// TIA Portal V15.1 export
// export: Created 2024-06-21T08:41:16.2567037Z, ExportSetting WithDefaults, DisplayName Totally Integrated Automation Portal, DisplayVersion V15.1 Update 5, DisplayName TIA Portal Openness, DisplayVersion V15.1 Update 5, DisplayName SINAMICS Startdrive Advanced, DisplayVersion V15.1, DisplayName G130, G150, S120, S150, SINAMICS MV, S210, DisplayVersion V15.1, DisplayName G110M, G120, G120C, G120D, G120P, DisplayVersion V15.1, DisplayName STEP 7 Professional, DisplayVersion V15.1 Update 5, DisplayName STEP 7 Safety, DisplayVersion V15.1, DisplayName WinCC Professional, DisplayVersion V15.1 Update 5, DisplayName SIMATIC Visualization Architect, DisplayVersion V15.1
FUNCTION_BLOCK "LGBRoller2W2S-MoviFitFCPN-S12B"   // FB6670, FBD
TITLE = LRoller2W2S-MoviFitFCPN / LGBRoller2W2S-MoviFitFCPN-S12B
{ S7_Optimized_Access := 'TRUE' }
AUTHOR : ENGIE
FAMILY : Transport
VERSION : 0.1
// =============================================================================
// This module is used in Applications when a roller one way two speed equipped 
// with SEW MOVIFIT-FC is needed. The roller can support single body tranport and 
// simultanious transport. The roller is equipped with a standard sensor setting, 
// one stop High Speed and one at the front for dual speed transport. The 
// roller uses standard handshaking signals to accomplish an infeed transfer 
// with the previous transport system and an outfeed with the next transport 
// system.
// The roller will support automatic Mode and manual Mode according specific 
// guidelines.
// The outfeed will be master over the infeed.
// Alarm "body not in Position" is also generated.
// All Alarms coming from sub-functions, TrfIn, TrfOut & LMotor2W2S-MoviFitFCPN or 
// from 
// local Alarm are summarized to give also the global Alarm A, B, C & D to 
// upper level.
// =============================================================================
// ============================================================================
// This module is used in Applications when a roller one way two speed equipped 
// with SEW MOVIFIT-FC is needed. The roller can support single body tranport and 
// simultanious transport. The roller is equipped with a standard sensor setting, 
// one stop High Speed and one at the front for dual speed transport. The 
// roller uses standard handshaking signals to accomplish an infeed transfer 
// with the previous transport system and an outfeed with the next transport 
// system.
// The roller will support automatic Mode and manual Mode according specific 
// guidelines.
// The outfeed will be master over the infeed.
// Alarm "body not in Position" is also generated.
// All Alarms coming from sub-functions, TrfIn, TrfOut & LMotor2W2S-MoviFitFCPN or 
// from 
// local Alarm are summarized to give also the global Alarm A, B, C & D to 
// upper level.
// ============================================================================
// stored: AutoNumber false, IsIECCheckEnabled false, IsRetainMemResEnabled false, MemoryReserve 100, SetENOAutomatically False, UDAEnableTagReadback false
   VAR_INPUT
      I_StopDetSet { ExternalAccessible := 'False'; ExternalVisible := 'False'; ExternalWritable := 'False'} : Bool;   // Stop detection set
      I_LowSpeedDetSet { ExternalAccessible := 'False'; ExternalVisible := 'False'; ExternalWritable := 'False'} : Bool;   // Lowspeed detection set
      I_StopDetRes { ExternalAccessible := 'False'; ExternalVisible := 'False'; ExternalWritable := 'False'} : Bool;   // Stop detection Reset
      I_LowSpeedDetRes { ExternalAccessible := 'False'; ExternalVisible := 'False'; ExternalWritable := 'False'} : Bool;   // Lowspeed stop detection Reset
      I_OccupiedDet { ExternalAccessible := 'False'; ExternalVisible := 'False'; ExternalWritable := 'False'} : Bool;   // Occupied detection
      I_TrfInSetBegin { ExternalAccessible := 'False'; ExternalVisible := 'False'; ExternalWritable := 'False'} : Bool;   // Load Begin: condition to start transfer IN set
      I_TrfInSetIntlkOk { ExternalAccessible := 'False'; ExternalVisible := 'False'; ExternalWritable := 'False'} : Bool;   // Transfer IN Interlock Set OK
      I_TrfInResBegin { ExternalAccessible := 'False'; ExternalVisible := 'False'; ExternalWritable := 'False'} : Bool;   // Load Begin: condition to start transfer IN Reset
      I_TrfInResIntlkOk { ExternalAccessible := 'False'; ExternalVisible := 'False'; ExternalWritable := 'False'} : Bool;   // Transfer IN Interlock Reset OKt
      I_TrfOutSetBegin { ExternalAccessible := 'False'; ExternalVisible := 'False'; ExternalWritable := 'False'} : Bool;   // Unload Begin: condition to start transfer OUT set
      I_TrfOutSetIntlkOk { ExternalAccessible := 'False'; ExternalVisible := 'False'; ExternalWritable := 'False'} : Bool;   // Transfer Out Interlock Set Ok
      I_TrfOutResBegin { ExternalAccessible := 'False'; ExternalVisible := 'False'; ExternalWritable := 'False'} : Bool;   // Unload Begin: condition to start transfer OUT Reset
      I_TrfOutResIntlkOk { ExternalAccessible := 'False'; ExternalVisible := 'False'; ExternalWritable := 'False'} : Bool;   // Transfer OUT Interlock Reset Ok
      I_TrfInSetRdyDlv { ExternalAccessible := 'False'; ExternalVisible := 'False'; ExternalWritable := 'False'} : Bool;   // Ready to deliver: Signal from previous object set
      I_TrfInSetTM { ExternalAccessible := 'False'; ExternalVisible := 'False'; ExternalWritable := 'False'} : Bool;   // Transfer busy signal from previous equipement set
      I_TrfOutSetRdyRcv { ExternalAccessible := 'False'; ExternalVisible := 'False'; ExternalWritable := 'False'} : Bool;   // Ready to Receive: Signal from next object set
      I_TrfOutSetArrived { ExternalAccessible := 'False'; ExternalVisible := 'False'; ExternalWritable := 'False'} : Bool;   // Body Arrived: Signal from next object Set
      I_TrfInResRdyDlv { ExternalAccessible := 'False'; ExternalVisible := 'False'; ExternalWritable := 'False'} : Bool;   // Ready to deliver: Signal from previous object Reset
      I_TrfInResTM { ExternalAccessible := 'False'; ExternalVisible := 'False'; ExternalWritable := 'False'} : Bool;   // Transfer busy signal from previous equipement Reset
      I_TrfOutResRdyRcv { ExternalAccessible := 'False'; ExternalVisible := 'False'; ExternalWritable := 'False'} : Bool;   // Ready to Receive: Signal from next object Reset
      I_TrfOutResArrived { ExternalAccessible := 'False'; ExternalVisible := 'False'; ExternalWritable := 'False'} : Bool;   // Body Arrived: Signal from next object Reset
      I_ManInfeedAllowedSet { ExternalAccessible := 'False'; ExternalVisible := 'False'; ExternalWritable := 'False'} : Bool;   // Manual Infeed Allowed Set (without PushButton)
      I_ManInfeedAllowedRes { ExternalAccessible := 'False'; ExternalVisible := 'False'; ExternalWritable := 'False'} : Bool;   // Manual Infeed Allowed Reset (without PushButton)
      I_ManLowSpdSel { ExternalAccessible := 'False'; ExternalVisible := 'False'; ExternalWritable := 'False'} : Bool;   // Low speed Selected in manual / Low speed Selected in manual by other roller
      I_ManHighSpdSel { ExternalAccessible := 'False'; ExternalVisible := 'False'; ExternalWritable := 'False'} : Bool;   // Low speed Selected in manual / High speed Selected in manual by other roller
      I_MotorProtection { ExternalAccessible := 'False'; ExternalVisible := 'False'; ExternalWritable := 'False'} : Bool;   // Motorprotection
      I_ReleaseBrake { ExternalAccessible := 'False'; ExternalVisible := 'False'; ExternalWritable := 'False'} : Bool;   // Release brake
      I_LocalPBSet { ExternalAccessible := 'False'; ExternalVisible := 'False'; ExternalWritable := 'False'} : Bool;   // Push button for manual movememt (on local panel)
      I_LocalPBRes { ExternalAccessible := 'False'; ExternalVisible := 'False'; ExternalWritable := 'False'} : Bool;   // Push button for manual movememt Reset(on local panel)
      I_BeltControlSetDet { ExternalAccessible := 'False'; ExternalVisible := 'False'; ExternalWritable := 'False'} : Bool;   // Sensor Belt Control Roller Set Direction
      I_BeltControlResDet { ExternalAccessible := 'False'; ExternalVisible := 'False'; ExternalWritable := 'False'} : Bool;   // Sensor Belt Control Roller Res Direction
      I_SafetyOk { ExternalAccessible := 'False'; ExternalVisible := 'False'; ExternalWritable := 'False'} : Bool;   // Safety Ok
      I_MotionStopOk { ExternalAccessible := 'False'; ExternalVisible := 'False'; ExternalWritable := 'False'} : Bool;   // Safety Ok / The motion stop is Ok
      I_LowSpeed { ExternalAccessible := 'False'; ExternalVisible := 'False'; ExternalWritable := 'False'} : Real;   // Low speed Value (set-up %)
      I_HighSpeed { ExternalAccessible := 'False'; ExternalVisible := 'False'; ExternalWritable := 'False'} : Real;   // High speed Value (set-up %)
      I_SafetyStatusWord1 { ExternalAccessible := 'False'; ExternalVisible := 'False'; ExternalWritable := 'False'} : Word;   // Safety Status / Safety Status Word
      I_SafetyStatusWord2 { ExternalAccessible := 'False'; ExternalVisible := 'False'; ExternalWritable := 'False'} : Word;   // Safety Status / Safety Status Word
      I_SafetyStatusWord3 { ExternalAccessible := 'False'; ExternalVisible := 'False'; ExternalWritable := 'False'} : Word;   // Safety Status / Safety Status Word
      I_SafetyControlWord1 { ExternalAccessible := 'False'; ExternalVisible := 'False'; ExternalWritable := 'False'} : Word;   // Safety Control Word
      I_SafetyControlWord2 { ExternalAccessible := 'False'; ExternalVisible := 'False'; ExternalWritable := 'False'} : Word;   // Safety Control Word
   END_VAR
   VAR_OUTPUT
      O_ReleaseBrake { ExternalAccessible := 'False'; ExternalVisible := 'False'; ExternalWritable := 'False'} : Bool;   // Release the brake of the Motor
      O_Active { ExternalAccessible := 'False'; ExternalVisible := 'False'; ExternalWritable := 'False'} : Bool;   // Roller is Active
      O_TrfInSetRdyRcv { ExternalAccessible := 'False'; ExternalVisible := 'False'; ExternalWritable := 'False'} : Bool;   // Ready to Receive: Signal to previous object set
      O_TrfInSetArrived { ExternalAccessible := 'False'; ExternalVisible := 'False'; ExternalWritable := 'False'} : Bool;   // Body Arrived: Signal to previous object Set
      O_TrfOutSetRdyDlv { ExternalAccessible := 'False'; ExternalVisible := 'False'; ExternalWritable := 'False'} : Bool;   // Ready to Deliver: Signal to next object set
      O_TrfOutSetTM { ExternalAccessible := 'False'; ExternalVisible := 'False'; ExternalWritable := 'False'} : Bool;   // Transfer: Signal to next object set
      O_TrfInResRdyRcv { ExternalAccessible := 'False'; ExternalVisible := 'False'; ExternalWritable := 'False'} : Bool;   // Ready to Receive: Signal to previous object Reset
      O_TrfInResArrived { ExternalAccessible := 'False'; ExternalVisible := 'False'; ExternalWritable := 'False'} : Bool;   // Body Arrived: Signal to previous object Reset
      O_TrfOutResRdyDlv { ExternalAccessible := 'False'; ExternalVisible := 'False'; ExternalWritable := 'False'} : Bool;   // Ready to Deliver: Signal to next object Reset
      O_TrfOutResTM { ExternalAccessible := 'False'; ExternalVisible := 'False'; ExternalWritable := 'False'} : Bool;   // Transfer: Signal to next object Reset
      O_TrfInSetActive { ExternalAccessible := 'False'; ExternalVisible := 'False'; ExternalWritable := 'False'} : Bool;   // Transfer in set active
      O_TrfInSetFinished { ExternalAccessible := 'False'; ExternalVisible := 'False'; ExternalWritable := 'False'} : Bool;   // Transfer in set finished
      O_TrfOutSetActive { ExternalAccessible := 'False'; ExternalVisible := 'False'; ExternalWritable := 'False'} : Bool;   // Transfer out set active
      O_TrfOutSetFinished { ExternalAccessible := 'False'; ExternalVisible := 'False'; ExternalWritable := 'False'} : Bool;   // Transfer out set finished
      O_TrfInResActive { ExternalAccessible := 'False'; ExternalVisible := 'False'; ExternalWritable := 'False'} : Bool;   // Transfer in Reset active
      O_TrfInResFinished { ExternalAccessible := 'False'; ExternalVisible := 'False'; ExternalWritable := 'False'} : Bool;   // Transfer in Reset finished
      O_TrfOutResActive { ExternalAccessible := 'False'; ExternalVisible := 'False'; ExternalWritable := 'False'} : Bool;   // Transfer out Reset active
      O_TrfOutResFinished { ExternalAccessible := 'False'; ExternalVisible := 'False'; ExternalWritable := 'False'} : Bool;   // Transfer out Reset finished
      O_BodyInPosition { ExternalAccessible := 'False'; ExternalVisible := 'False'; ExternalWritable := 'False'} : Bool;   // Body in Position on roller
      O_ManLowSpdSel { ExternalAccessible := 'False'; ExternalVisible := 'False'; ExternalWritable := 'False'} : Bool;   // Low speed Selected in manual
      O_ManHighSpdSel { ExternalAccessible := 'False'; ExternalVisible := 'False'; ExternalWritable := 'False'} : Bool;   // Low speed Selected in manual / High speed Selected in manual
      O_LedRoller { ExternalAccessible := 'False'; ExternalVisible := 'False'; ExternalWritable := 'False'} : Bool;   // Led of roller
      O_LSpdSetMotorCmd { ExternalAccessible := 'False'; ExternalVisible := 'False'; ExternalWritable := 'False'} : Bool;   // Low Speed Set Command from function after Interlock
      O_HSpdSetMotorCmd { ExternalAccessible := 'False'; ExternalVisible := 'False'; ExternalWritable := 'False'} : Bool;   // High Speed Set Command from function after Interlock
      O_LSpdResMotorCmd { ExternalAccessible := 'False'; ExternalVisible := 'False'; ExternalWritable := 'False'} : Bool;   // Low speed Reset Command from function after Interlock
      O_HSpdResMotorCmd { ExternalAccessible := 'False'; ExternalVisible := 'False'; ExternalWritable := 'False'} : Bool;   // High speed Reset Command from function after Interlock
      O_AlarmABCondition { ExternalAccessible := 'False'; ExternalVisible := 'False'; ExternalWritable := 'False'} : Bool;   // Alarm AB Condition
      O_AlarmA { ExternalAccessible := 'False'; ExternalVisible := 'False'; ExternalWritable := 'False'} : Bool;   // Alarm A
      O_AlarmB { ExternalAccessible := 'False'; ExternalVisible := 'False'; ExternalWritable := 'False'} : Bool;   // Alarm B
      O_AlarmC { ExternalAccessible := 'False'; ExternalVisible := 'False'; ExternalWritable := 'False'} : Bool;   // Alarm C
      O_AlarmD { ExternalAccessible := 'False'; ExternalVisible := 'False'; ExternalWritable := 'False'} : Bool;   // Alarm D
      O_Occupied { ExternalAccessible := 'False'; ExternalVisible := 'False'; ExternalWritable := 'False'} : Bool;   // Roller Occupied
      H_AlarmDWord { ExternalAccessible := 'False'; ExternalVisible := 'False'; ExternalWritable := 'False'} : DWord;   // Alarm Word
   END_VAR
   VAR_IN_OUT
      IO_Modes : "Modes";   // Modes
      H_HMI : "H_HMI";   // Animation
      "H_GBRoller2W2S-MoviFitFCPN-S12B" : "H_GBRoller2W2S-MoviFitFCPN-S12B";   // Animation
      C_RollerConvConfig : "RollerConvMoviFitFCPNConfig";   // Config
   END_VAR
   VAR
      _LTrfInSet { ExternalAccessible := 'False'; ExternalVisible := 'False'; ExternalWritable := 'False'} : "LGBTrfIn";   // FB
      _LTrfOutSet { ExternalAccessible := 'False'; ExternalVisible := 'False'; ExternalWritable := 'False'} : "LGBTrfOut";   // FB
      _LTrfInRes { ExternalAccessible := 'False'; ExternalVisible := 'False'; ExternalWritable := 'False'} : "LGBTrfIn";   // FB
      _LTrfOutRes { ExternalAccessible := 'False'; ExternalVisible := 'False'; ExternalWritable := 'False'} : "LGBTrfOut";   // FB
      _Motor { ExternalAccessible := 'False'; ExternalVisible := 'False'; ExternalWritable := 'False'} : "LGBMotor2W2S-MoviFitFCPN-S12B";   // FB
      AB_BeltControlSetDet { ExternalAccessible := 'False'; ExternalVisible := 'False'; ExternalWritable := 'False'} : Bool;   // Belt Check Roller Set Direction
      AB_BeltControlResDet { ExternalAccessible := 'False'; ExternalVisible := 'False'; ExternalWritable := 'False'} : Bool;   // Belt Check Roller Reset Direction
      AC_BodyNotInPos { ExternalAccessible := 'False'; ExternalVisible := 'False'; ExternalWritable := 'False'} : Bool;   // Body, Skid Not In Position
      AD_TrfInResInterlock { ExternalAccessible := 'False'; ExternalVisible := 'False'; ExternalWritable := 'False'} : Bool;   // Interlock Not Ok Transport In Reset
      AB_TrfOutSetOverTime { ExternalAccessible := 'False'; ExternalVisible := 'False'; ExternalWritable := 'False'} : Bool;   // Timeout Set
      AD_TrfOutSetInterlock { ExternalAccessible := 'False'; ExternalVisible := 'False'; ExternalWritable := 'False'} : Bool;   // Interlock Not Ok Transport Out Set
      AD_TrfInSetInterlock { ExternalAccessible := 'False'; ExternalVisible := 'False'; ExternalWritable := 'False'} : Bool;   // Interlock Not Ok Transport In Set
      AB_TrfOutResOverTime { ExternalAccessible := 'False'; ExternalVisible := 'False'; ExternalWritable := 'False'} : Bool;   // Timeout Reset
      AD_TrfOutResInterlock { ExternalAccessible := 'False'; ExternalVisible := 'False'; ExternalWritable := 'False'} : Bool;   // Interlock Not Ok Transport Out Reset
      AB_LSpeedDetMissing { ExternalAccessible := 'False'; ExternalVisible := 'False'; ExternalWritable := 'False'} : Bool;   // Low Speed Detector Missing
      AA_MotorProtection { ExternalAccessible := 'False'; ExternalVisible := 'False'; ExternalWritable := 'False'} : Bool;   // Motorprotection Tripped / Motor Protection Tripped
      AA_SafetySwitch { ExternalAccessible := 'False'; ExternalVisible := 'False'; ExternalWritable := 'False'} : Bool;   // Safety Switch Not Ok
      AB_STO { ExternalAccessible := 'False'; ExternalVisible := 'False'; ExternalWritable := 'False'} : Bool;   // Safety Switch Not Ok / Safety output to drive is active but no response from drive that the safety is ok
      AD_Warning { ExternalAccessible := 'False'; ExternalVisible := 'False'; ExternalWritable := 'False'} : Bool;   // Frequency Control
      AA_NoBusControl { ExternalAccessible := 'False'; ExternalVisible := 'False'; ExternalWritable := 'False'} : Bool;   // Frequency Control / Bus control inactive / Frekvensstyrning
      AB_Alarm { ExternalAccessible := 'False'; ExternalVisible := 'False'; ExternalWritable := 'False'} : Bool;   // Frequency Control
      AC_TrfInStopped { ExternalAccessible := 'False'; ExternalVisible := 'False'; ExternalWritable := 'False'} : Bool;   // Transfer In Stopped
      AC_StopDetSet { ExternalAccessible := 'False'; ExternalVisible := 'False'; ExternalWritable := 'False'} : Bool;   // Body, Skid Not In Position Stop Det Set
      AC_StopDetRes { ExternalAccessible := 'False'; ExternalVisible := 'False'; ExternalWritable := 'False'} : Bool;   // Body, Skid Not In Position Stop Det Reset
      AC_LowSpdDetSet { ExternalAccessible := 'False'; ExternalVisible := 'False'; ExternalWritable := 'False'} : Bool;   // Body, Skid Not In Position Low Speed Det Set
      AC_LowSpdDetRes { ExternalAccessible := 'False'; ExternalVisible := 'False'; ExternalWritable := 'False'} : Bool;   // Body, Skid Not In Position Low Speed Det Reset
      AD_MotionStop { ExternalAccessible := 'False'; ExternalVisible := 'False'; ExternalWritable := 'False'} : Bool;   // Motion Stop
      AC_ConfigCalibrationAlm { ExternalAccessible := 'False'; ExternalVisible := 'False'; ExternalWritable := 'False'} : Bool;   // The Config values for Alarm Transfer time must be ALL zero or ALL different from zero
      AD_CalibrationSetWarn { ExternalAccessible := 'False'; ExternalVisible := 'False'; ExternalWritable := 'False'} : Bool;   // No High speed selected so Calibration is not possible for SET direction
      AD_CalibrationResetWarn { ExternalAccessible := 'False'; ExternalVisible := 'False'; ExternalWritable := 'False'} : Bool;   // No High speed selected so Calibration is not possible for RESET direction
      AC_ConfigRampAlm { ExternalAccessible := 'False'; ExternalVisible := 'False'; ExternalWritable := 'False'} : Bool;   // The config value for the ramp is not correct, must be zero or the config values for the calculation of the ramp must be ALL zero
      AC_ConfigRampCalcAlm { ExternalAccessible := 'False'; ExternalVisible := 'False'; ExternalWritable := 'False'} : Bool;   // The config values for the calculation of the ramp must be ALL different from zero
      PODataNotEnabled { ExternalAccessible := 'False'; ExternalVisible := 'False'; ExternalWritable := 'False'} : Bool;   // Bus control inactive
      SafetyOk { ExternalAccessible := 'False'; ExternalVisible := 'False'; ExternalWritable := 'False'} : Bool;   // Safety Ok
   END_VAR
   VAR RETAIN
      LowSpeedSetDetOk { ExternalAccessible := 'False'; ExternalVisible := 'False'; ExternalWritable := 'False'} : Bool;   // Low speed detector set ok
      LowSpeedResDetOk { ExternalAccessible := 'False'; ExternalVisible := 'False'; ExternalWritable := 'False'} : Bool;   // Low speed detector Reset ok
   END_VAR
   VAR
      AllDet { ExternalAccessible := 'False'; ExternalVisible := 'False'; ExternalWritable := 'False'} : Bool;   // AND of all detections
      AnyDet { ExternalAccessible := 'False'; ExternalVisible := 'False'; ExternalWritable := 'False'} : Bool;   // OR of all detections
      MotorLoopActive { ExternalAccessible := 'False'; ExternalVisible := 'False'; ExternalWritable := 'False'} : Bool;   // Motor Loop Active
      TrfInSetIntlkOk { ExternalAccessible := 'False'; ExternalVisible := 'False'; ExternalWritable := 'False'} : Bool;   // Transfer IN Interlock Set OK
      TrfInResIntlkOk { ExternalAccessible := 'False'; ExternalVisible := 'False'; ExternalWritable := 'False'} : Bool;   // Transfer IN Interlock Reset OKt / Transfer IN Interlock Reset OK
      TrfOutResIntlkOk { ExternalAccessible := 'False'; ExternalVisible := 'False'; ExternalWritable := 'False'} : Bool;   // Transfer OUT Interlock Reset Ok
      TrfOutSetIntlkOk { ExternalAccessible := 'False'; ExternalVisible := 'False'; ExternalWritable := 'False'} : Bool;   // Transfer Out Interlock Set Ok
      TrfInResCmd { ExternalAccessible := 'False'; ExternalVisible := 'False'; ExternalWritable := 'False'} : Bool;   // Command after Interlock to Motor Reset
      TrfInfeedHoldSet { ExternalAccessible := 'False'; ExternalVisible := 'False'; ExternalWritable := 'False'} : Bool;   // Transfer infeed hold set direction
      TrfOutSetCmd { ExternalAccessible := 'False'; ExternalVisible := 'False'; ExternalWritable := 'False'} : Bool;   // Command after Interlock to Motor set
      TrfOutfeedHoldSet { ExternalAccessible := 'False'; ExternalVisible := 'False'; ExternalWritable := 'False'} : Bool;   // Transfer outfeed hold set direction
      TrfInSetCmd { ExternalAccessible := 'False'; ExternalVisible := 'False'; ExternalWritable := 'False'} : Bool;   // Command after Interlock to Motor set
      TrfInfeedHoldRes { ExternalAccessible := 'False'; ExternalVisible := 'False'; ExternalWritable := 'False'} : Bool;   // Transfer infeed hold Reset direction
      TrfOutResCmd { ExternalAccessible := 'False'; ExternalVisible := 'False'; ExternalWritable := 'False'} : Bool;   // Command after Interlock to Motor Reset
      TrfOutfeedHoldRes { ExternalAccessible := 'False'; ExternalVisible := 'False'; ExternalWritable := 'False'} : Bool;   // Transfer outfeed hold Reset direction
      MotorCmdLSpdSet { ExternalAccessible := 'False'; ExternalVisible := 'False'; ExternalWritable := 'False'} : Bool;   // Command to Motorloop low Speed Set
      MotorCmdLSpdRes { ExternalAccessible := 'False'; ExternalVisible := 'False'; ExternalWritable := 'False'} : Bool;   // Command to Motorloop low speed Reset
      MotorCmdHSpdSet { ExternalAccessible := 'False'; ExternalVisible := 'False'; ExternalWritable := 'False'} : Bool;   // Command to Motorloop High Speed Set
      MotorCmdHSpdRes { ExternalAccessible := 'False'; ExternalVisible := 'False'; ExternalWritable := 'False'} : Bool;   // Command to Motorloop High Speed Reset
   END_VAR
   VAR RETAIN
      LowSpeedDetSetMem { ExternalAccessible := 'False'; ExternalVisible := 'False'; ExternalWritable := 'False'} : Bool;   // Memorisation stop High Speed Set direction
      LowSpeedDetResMem { ExternalAccessible := 'False'; ExternalVisible := 'False'; ExternalWritable := 'False'} : Bool;   // Memorisation stop high peed Reset direction
   END_VAR
   VAR
      TrfInSetActive { ExternalAccessible := 'False'; ExternalVisible := 'False'; ExternalWritable := 'False'} : Bool;   // Load Active Set
      TrfOutSetActive { ExternalAccessible := 'False'; ExternalVisible := 'False'; ExternalWritable := 'False'} : Bool;   // Unload active Set
      TrfOutSetFinished { ExternalAccessible := 'False'; ExternalVisible := 'False'; ExternalWritable := 'False'} : Bool;   // Unload finished Set
      TrfInResActive { ExternalAccessible := 'False'; ExternalVisible := 'False'; ExternalWritable := 'False'} : Bool;   // Load Active Reset
      TrfOutResActive { ExternalAccessible := 'False'; ExternalVisible := 'False'; ExternalWritable := 'False'} : Bool;   // Unload active Reset
      TrfOutResFinished { ExternalAccessible := 'False'; ExternalVisible := 'False'; ExternalWritable := 'False'} : Bool;   // Unload finished Reset
      StationOnly { ExternalAccessible := 'False'; ExternalVisible := 'False'; ExternalWritable := 'False'} : Bool;   // Station Only
      AlarmA { ExternalAccessible := 'False'; ExternalVisible := 'False'; ExternalWritable := 'False'} : Bool;   // Alarm A
      AlarmB { ExternalAccessible := 'False'; ExternalVisible := 'False'; ExternalWritable := 'False'} : Bool;   // Alarm B
      AlarmC { ExternalAccessible := 'False'; ExternalVisible := 'False'; ExternalWritable := 'False'} : Bool;   // Alarm C
      AlarmD { ExternalAccessible := 'False'; ExternalVisible := 'False'; ExternalWritable := 'False'} : Bool;   // Alarm D
      AlarmABCondition { ExternalAccessible := 'False'; ExternalVisible := 'False'; ExternalWritable := 'False'} : Bool;   // Alarm AB Condition
      ManLowSpdSel { ExternalAccessible := 'False'; ExternalVisible := 'False'; ExternalWritable := 'False'} : Bool;   // Low speed Selected in manual
      BodyInPosition { ExternalAccessible := 'False'; ExternalVisible := 'False'; ExternalWritable := 'False'} : Bool;   // Body in Position
      TrfInResRdyRcv { ExternalAccessible := 'False'; ExternalVisible := 'False'; ExternalWritable := 'False'} : Bool;   // Ready to Receive: Signal to previous object Reset
      TrfInResArrived { ExternalAccessible := 'False'; ExternalVisible := 'False'; ExternalWritable := 'False'} : Bool;   // Body Arrived: Signal to previous object Reset
      TrfInResFinished { ExternalAccessible := 'False'; ExternalVisible := 'False'; ExternalWritable := 'False'} : Bool;   // Body Arrived: Signal to TrfOut module Reset (Reset TrfOutCmd)
      TrfOutSetRdyDlv { ExternalAccessible := 'False'; ExternalVisible := 'False'; ExternalWritable := 'False'} : Bool;   // Ready to Deliver: Signal to next object set
      TrfOutSetTM { ExternalAccessible := 'False'; ExternalVisible := 'False'; ExternalWritable := 'False'} : Bool;   // Transfer : Signal transfer memory to next object set
      TrfInSetTrfOutSetTM { ExternalAccessible := 'False'; ExternalVisible := 'False'; ExternalWritable := 'False'} : Bool;   // Transfer memory set
      TrfInSetRdyRcv { ExternalAccessible := 'False'; ExternalVisible := 'False'; ExternalWritable := 'False'} : Bool;   // Ready to Receive: Signal to previous object set
      TrfInSetArrived { ExternalAccessible := 'False'; ExternalVisible := 'False'; ExternalWritable := 'False'} : Bool;   // Body Arrived: Signal to previous object Set
      TrfInSetFinished { ExternalAccessible := 'False'; ExternalVisible := 'False'; ExternalWritable := 'False'} : Bool;   // Body Arrived: Signal to TrfOut module set (Reset TrfOutCmd)
      StopTrfOutSetCmd { ExternalAccessible := 'False'; ExternalVisible := 'False'; ExternalWritable := 'False'} : Bool;   // Body Arrived: Signal to previous object Set
      TrfOutResRdyDlv { ExternalAccessible := 'False'; ExternalVisible := 'False'; ExternalWritable := 'False'} : Bool;   // Ready to Deliver: Signal to next object Reset
      TrfOutResTM { ExternalAccessible := 'False'; ExternalVisible := 'False'; ExternalWritable := 'False'} : Bool;   // Transfer : Signal transfer memory to next object Reset
      TrfInResTrfOutResTM { ExternalAccessible := 'False'; ExternalVisible := 'False'; ExternalWritable := 'False'} : Bool;   // Transfer memory Reset
      MotorLoopAlarmCond { ExternalAccessible := 'False'; ExternalVisible := 'False'; ExternalWritable := 'False'} : Bool;   // Motor loop Alarm condition
      TrfOutResAlmCond { ExternalAccessible := 'False'; ExternalVisible := 'False'; ExternalWritable := 'False'} : Bool;   // TrfOut Alarm condition
      TrfOutSetAlmCond { ExternalAccessible := 'False'; ExternalVisible := 'False'; ExternalWritable := 'False'} : Bool;   // TrfOut Alarm condition
      StopTrfOutResCmd { ExternalAccessible := 'False'; ExternalVisible := 'False'; ExternalWritable := 'False'} : Bool;   // Body Arrived: Signal to previous object Reset
      LowSpeedDetMisingCond { ExternalAccessible := 'False'; ExternalVisible := 'False'; ExternalWritable := 'False'} : Bool;   // Low speed detector misiing condition
      ReleaseBrake { ExternalAccessible := 'False'; ExternalVisible := 'False'; ExternalWritable := 'False'} : Bool;   // Release brake
      ReadyForOperation { ExternalAccessible := 'False'; ExternalVisible := 'False'; ExternalWritable := 'False'} : Bool;   // Ready for operation
      BeltControlSetAlarmABCondition { ExternalAccessible := 'False'; ExternalVisible := 'False'; ExternalWritable := 'False'} : Bool;   // Belt Control AB Condition
      BeltControlResAlarmABCondition { ExternalAccessible := 'False'; ExternalVisible := 'False'; ExternalWritable := 'False'} : Bool;   // Belt Control AB Condition
      _BeltControlSet { ExternalAccessible := 'False'; ExternalVisible := 'False'; ExternalWritable := 'False'} : "L1AlarmMultiIn";   // FB
      _BeltControlRes { ExternalAccessible := 'False'; ExternalVisible := 'False'; ExternalWritable := 'False'} : "L1AlarmMultiIn";   // FB
      BeltPulseCountSet { ExternalAccessible := 'False'; ExternalVisible := 'False'; ExternalWritable := 'False'} : DInt;   // Temp
      BeltPulseCountRes { ExternalAccessible := 'False'; ExternalVisible := 'False'; ExternalWritable := 'False'} : DInt;   // Temp
      _InitBeltCntSet { ExternalAccessible := 'False'; ExternalVisible := 'False'; ExternalWritable := 'False'} : "LChangeOfState";   // FB
      _InitBeltCntRes { ExternalAccessible := 'False'; ExternalVisible := 'False'; ExternalWritable := 'False'} : "LChangeOfState";   // FB
      BeltPosEdgeSet1 { ExternalAccessible := 'False'; ExternalVisible := 'False'; ExternalWritable := 'False'} : Bool;   // Pos Edge
      BeltPosEdgeSet2 { ExternalAccessible := 'False'; ExternalVisible := 'False'; ExternalWritable := 'False'} : Bool;   // Pos Edge
      BeltPosEdgeRes1 { ExternalAccessible := 'False'; ExternalVisible := 'False'; ExternalWritable := 'False'} : Bool;   // Pos Edge
      BeltPosEdgeRes2 { ExternalAccessible := 'False'; ExternalVisible := 'False'; ExternalWritable := 'False'} : Bool;   // Pos Edge
      InitBeltCounterSet { ExternalAccessible := 'False'; ExternalVisible := 'False'; ExternalWritable := 'False'} : Bool;   // Init
      InitBeltCounterRes { ExternalAccessible := 'False'; ExternalVisible := 'False'; ExternalWritable := 'False'} : Bool;   // Init
      _StationOnly { ExternalAccessible := 'False'; ExternalVisible := 'False'; ExternalWritable := 'False'} : "LToggle";   // FB
      _NoTrfIn { ExternalAccessible := 'False'; ExternalVisible := 'False'; ExternalWritable := 'False'} : "LToggle";   // FB
      Edge { ExternalAccessible := 'False'; ExternalVisible := 'False'; ExternalWritable := 'False'} : Array[1..7] of Bool;   // Edge
   END_VAR
   VAR_TEMP
      NotUsedH_HMI : "H_HMI";   // Temp
      H_HMITrfInSet : "H_HMI";   // Temp
      H_HMITrfInRes : "H_HMI";   // Temp
      H_HMITrfOutSet : "H_HMI";   // Temp
      H_HMITrfOutRes : "H_HMI";   // Temp
      H_HMIMotor : "H_HMI";   // Temp
      HMICMD : "ConvHMICMD";   // Temp
      TempDInt : DInt;   // Temp DInt
   END_VAR
   VAR_TEMP   // added for the SCL form of the ladder/FBD networks
      _w1 : Bool;
      _w2 : Bool;
      _w3 : Bool;
      _w4 : Bool;
   END_VAR
BEGIN

REGION Network 1: **** 1 - Inputs **** HMI Commands
   // HMI Commands
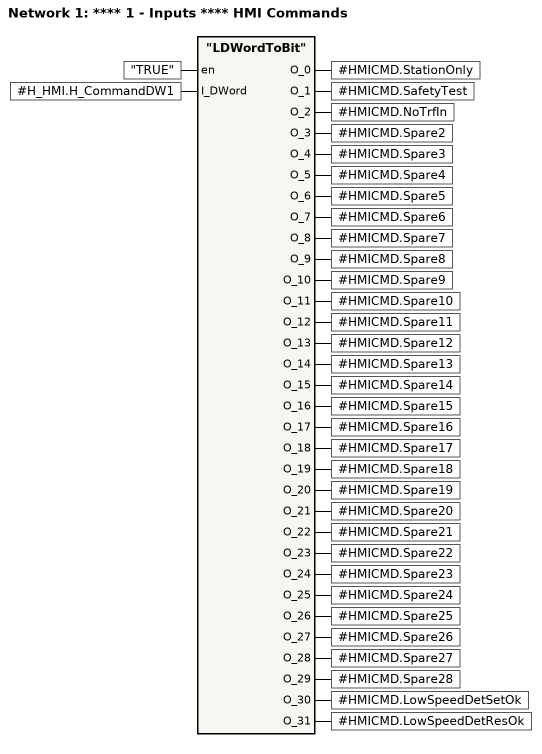
   IF "TRUE" THEN
       "LDWordToBit"(I_DWord := #H_HMI.H_CommandDW1,
                     O_0 => #HMICMD.StationOnly,
                     O_1 => #HMICMD.SafetyTest,
                     O_2 => #HMICMD.NoTrfIn,
                     O_3 => #HMICMD.Spare2,
                     O_4 => #HMICMD.Spare3,
                     O_5 => #HMICMD.Spare4,
                     O_6 => #HMICMD.Spare5,
                     O_7 => #HMICMD.Spare6,
                     O_8 => #HMICMD.Spare7,
                     O_9 => #HMICMD.Spare8,
                     O_10 => #HMICMD.Spare9,
                     O_11 => #HMICMD.Spare10,
                     O_12 => #HMICMD.Spare11,
                     O_13 => #HMICMD.Spare12,
                     O_14 => #HMICMD.Spare13,
                     O_15 => #HMICMD.Spare14,
                     O_16 => #HMICMD.Spare15,
                     O_17 => #HMICMD.Spare16,
                     O_18 => #HMICMD.Spare17,
                     O_19 => #HMICMD.Spare18,
                     O_20 => #HMICMD.Spare19,
                     O_21 => #HMICMD.Spare20,
                     O_22 => #HMICMD.Spare21,
                     O_23 => #HMICMD.Spare22,
                     O_24 => #HMICMD.Spare23,
                     O_25 => #HMICMD.Spare24,
                     O_26 => #HMICMD.Spare25,
                     O_27 => #HMICMD.Spare26,
                     O_28 => #HMICMD.Spare27,
                     O_29 => #HMICMD.Spare28,
                     O_30 => #HMICMD.LowSpeedDetSetOk,
                     O_31 => #HMICMD.LowSpeedDetResOk);
   END_IF;
END_REGION

REGION Network 2: **** 1 - Inputs **** AND of all detections
   // AND of all detections
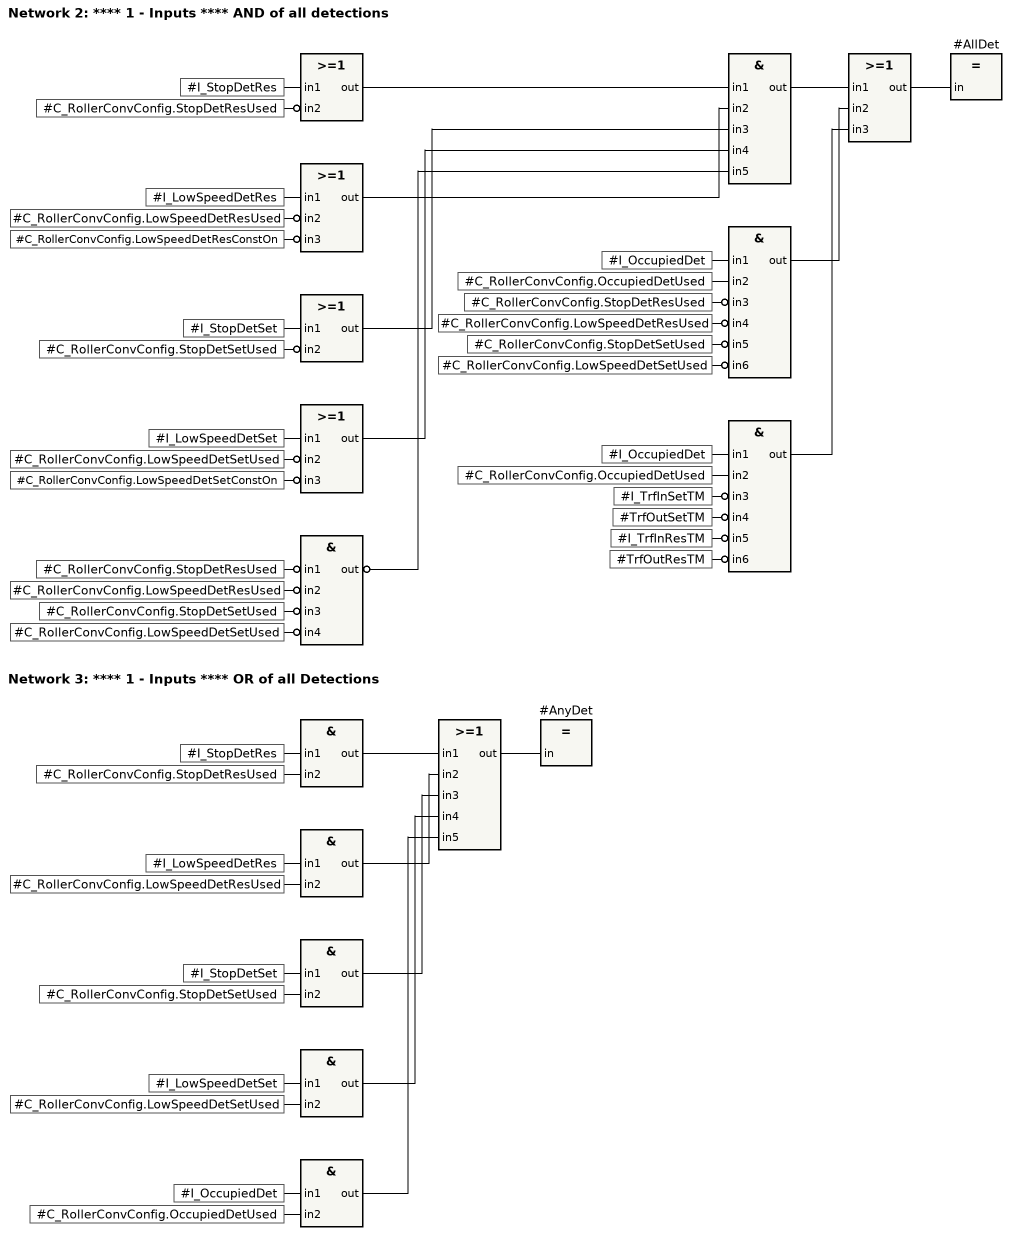
   #AllDet := ((#I_StopDetRes OR NOT #C_RollerConvConfig.StopDetResUsed) AND (#I_LowSpeedDetRes OR NOT #C_RollerConvConfig.LowSpeedDetResUsed OR NOT #C_RollerConvConfig.LowSpeedDetResConstOn) AND (#I_StopDetSet OR NOT #C_RollerConvConfig.StopDetSetUsed) AND (#I_LowSpeedDetSet OR NOT #C_RollerConvConfig.LowSpeedDetSetUsed OR NOT #C_RollerConvConfig.LowSpeedDetSetConstOn) AND NOT (NOT #C_RollerConvConfig.StopDetResUsed AND NOT #C_RollerConvConfig.LowSpeedDetResUsed AND NOT #C_RollerConvConfig.StopDetSetUsed AND NOT #C_RollerConvConfig.LowSpeedDetSetUsed)) OR (#I_OccupiedDet AND #C_RollerConvConfig.OccupiedDetUsed AND NOT #C_RollerConvConfig.StopDetResUsed AND NOT #C_RollerConvConfig.LowSpeedDetResUsed AND NOT #C_RollerConvConfig.StopDetSetUsed AND NOT #C_RollerConvConfig.LowSpeedDetSetUsed) OR (#I_OccupiedDet AND #C_RollerConvConfig.OccupiedDetUsed AND NOT #I_TrfInSetTM AND NOT #TrfOutSetTM AND NOT #I_TrfInResTM AND NOT #TrfOutResTM);
END_REGION

REGION Network 3: **** 1 - Inputs **** OR of all Detections
   // OR of all Detections
   #AnyDet := (#I_StopDetRes AND #C_RollerConvConfig.StopDetResUsed) OR (#I_LowSpeedDetRes AND #C_RollerConvConfig.LowSpeedDetResUsed) OR (#I_StopDetSet AND #C_RollerConvConfig.StopDetSetUsed) OR (#I_LowSpeedDetSet AND #C_RollerConvConfig.LowSpeedDetSetUsed) OR (#I_OccupiedDet AND #C_RollerConvConfig.OccupiedDetUsed);
END_REGION

REGION Network 4: **** 1 - Inputs **** Low speed detector been on
   // Low speed detector been on
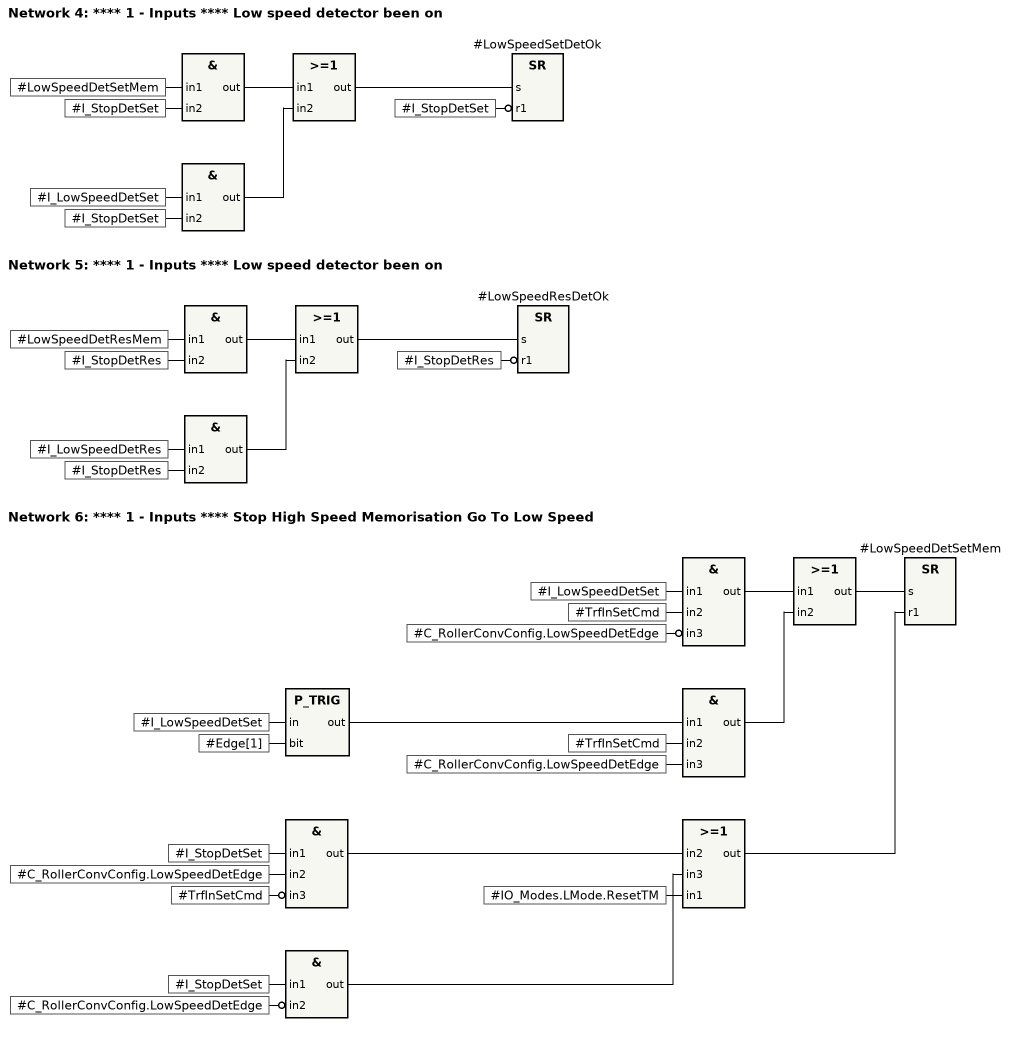
   IF (#LowSpeedDetSetMem AND #I_StopDetSet) OR (#I_LowSpeedDetSet AND #I_StopDetSet) THEN
       #LowSpeedSetDetOk := TRUE;   // SR flip-flop
   END_IF;
   IF NOT #I_StopDetSet THEN #LowSpeedSetDetOk := FALSE; END_IF;
END_REGION

REGION Network 5: **** 1 - Inputs **** Low speed detector been on
   // Low speed detector been on
   IF (#LowSpeedDetResMem AND #I_StopDetRes) OR (#I_LowSpeedDetRes AND #I_StopDetRes) THEN
       #LowSpeedResDetOk := TRUE;   // SR flip-flop
   END_IF;
   IF NOT #I_StopDetRes THEN #LowSpeedResDetOk := FALSE; END_IF;
END_REGION

REGION Network 6: **** 1 - Inputs **** Stop High Speed Memorisation Go To Low Speed
   // Stop High Speed Memorisation Go To Low Speed
   #_w1 := #I_LowSpeedDetSet AND NOT #Edge[1];   // rising edge
   #Edge[1] := #I_LowSpeedDetSet;
   IF (#I_LowSpeedDetSet AND #TrfInSetCmd AND NOT #C_RollerConvConfig.LowSpeedDetEdge) OR (#_w1 AND #TrfInSetCmd AND #C_RollerConvConfig.LowSpeedDetEdge) THEN
       #LowSpeedDetSetMem := TRUE;   // SR flip-flop
   END_IF;
   IF (#I_StopDetSet AND #C_RollerConvConfig.LowSpeedDetEdge AND NOT #TrfInSetCmd) OR (#I_StopDetSet AND NOT #C_RollerConvConfig.LowSpeedDetEdge) OR #IO_Modes.LMode.ResetTM THEN
       #LowSpeedDetSetMem := FALSE;
   END_IF;
END_REGION

REGION Network 7: **** 1 - Inputs **** Stop High Speed Memorisation Go To Low Speed
   // Stop High Speed Memorisation Go To Low Speed
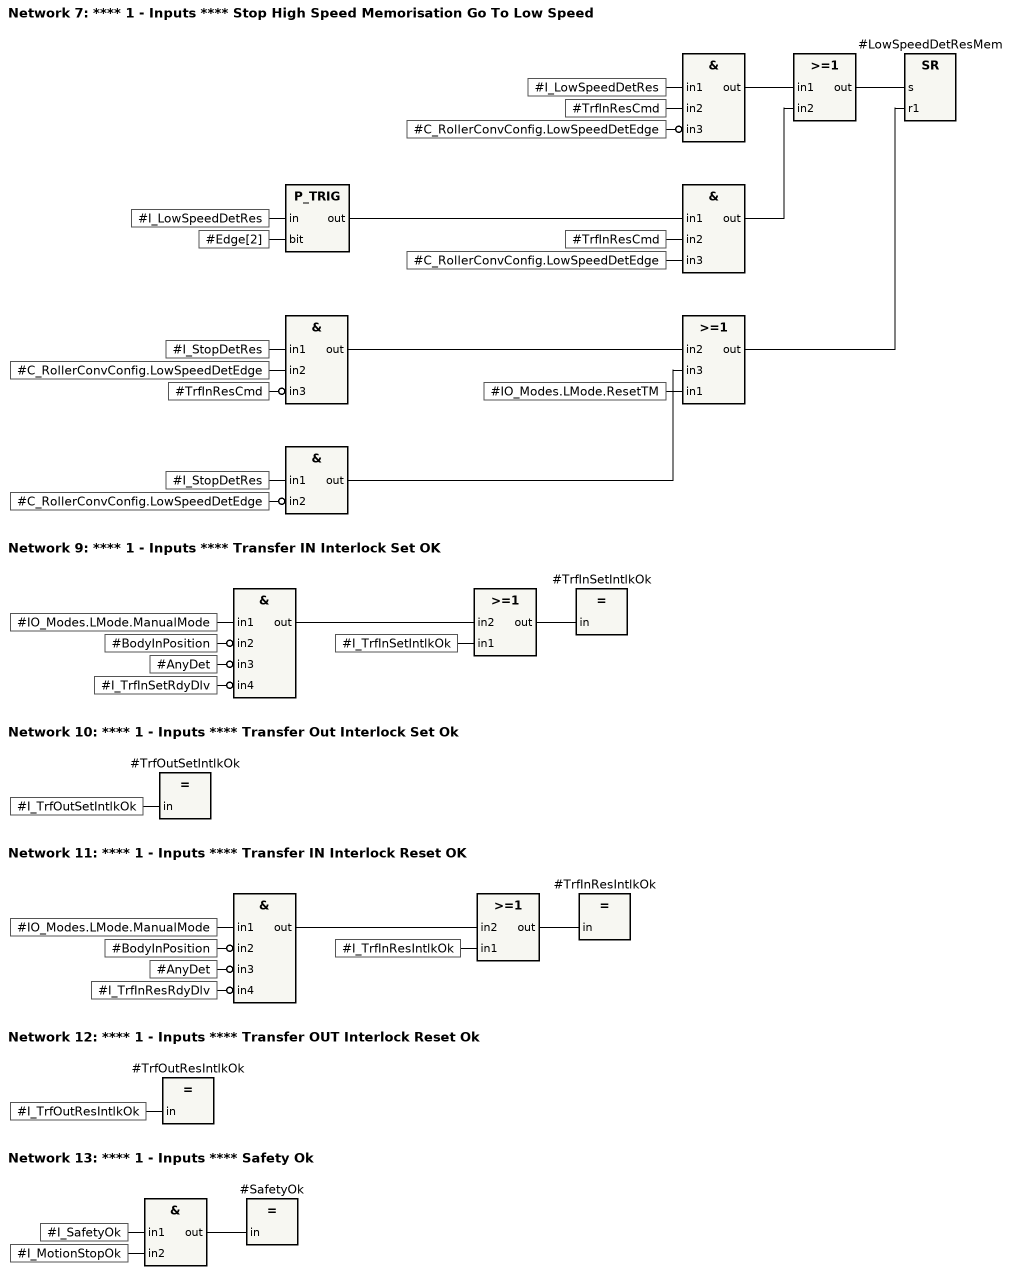
   #_w1 := #I_LowSpeedDetRes AND NOT #Edge[2];   // rising edge
   #Edge[2] := #I_LowSpeedDetRes;
   IF (#I_LowSpeedDetRes AND #TrfInResCmd AND NOT #C_RollerConvConfig.LowSpeedDetEdge) OR (#_w1 AND #TrfInResCmd AND #C_RollerConvConfig.LowSpeedDetEdge) THEN
       #LowSpeedDetResMem := TRUE;   // SR flip-flop
   END_IF;
   IF (#I_StopDetRes AND #C_RollerConvConfig.LowSpeedDetEdge AND NOT #TrfInResCmd) OR (#I_StopDetRes AND NOT #C_RollerConvConfig.LowSpeedDetEdge) OR #IO_Modes.LMode.ResetTM THEN
       #LowSpeedDetResMem := FALSE;
   END_IF;
END_REGION

NETWORK
TITLE = **** 1 - Inputs **** Init Belt Control Set And Reset Direction
// Init Belt Control Set And Reset Direction
      CALL  #_InitBeltCntSet
      ( I_In     := #I_BeltControlSetDet,
        O_OutPut := #InitBeltCounterSet
      );
      NOP   0;

      CALL  #_InitBeltCntRes
      ( I_In     := #I_BeltControlResDet,
        O_OutPut := #InitBeltCounterRes
      );
      NOP   0;

      A(;
      O     #InitBeltCounterSet;
      O;
//      A     #ManualMode AP
      A     #IO_Modes.LMode.AlarmResetPB;
      );
      JCN   NCSet;
      L     0;
      T     #BeltPulseCountSet;
NCSet:NOP   0;

      A(;
      O     #InitBeltCounterRes;
      O;
//  A     #ManualMode AP
      A     #IO_Modes.LMode.AlarmResetPB;
      );
      JCN   NCReset;
      L     0;
      T     #BeltPulseCountRes;
NCReset:NOP   0;


REGION Network 9: **** 1 - Inputs **** Transfer IN Interlock Set OK
   #TrfInSetIntlkOk := (#IO_Modes.LMode.ManualMode AND NOT #BodyInPosition AND NOT #AnyDet AND NOT #I_TrfInSetRdyDlv) OR #I_TrfInSetIntlkOk;
END_REGION

REGION Network 10: **** 1 - Inputs **** Transfer Out Interlock Set Ok
   #TrfOutSetIntlkOk := #I_TrfOutSetIntlkOk;
END_REGION

REGION Network 11: **** 1 - Inputs **** Transfer IN Interlock Reset OK
   #TrfInResIntlkOk := (#IO_Modes.LMode.ManualMode AND NOT #BodyInPosition AND NOT #AnyDet AND NOT #I_TrfInResRdyDlv) OR #I_TrfInResIntlkOk;
END_REGION

REGION Network 12: **** 1 - Inputs **** Transfer OUT Interlock Reset Ok
   #TrfOutResIntlkOk := #I_TrfOutResIntlkOk;
END_REGION

REGION Network 13: **** 1 - Inputs **** Safety Ok
   #SafetyOk := #I_SafetyOk AND #I_MotionStopOk;
END_REGION

REGION Network 14: **** 2.2 - Alarms - Alarm Generation **** Alarm Body Not In Position
   // Alarm Body Not In Position
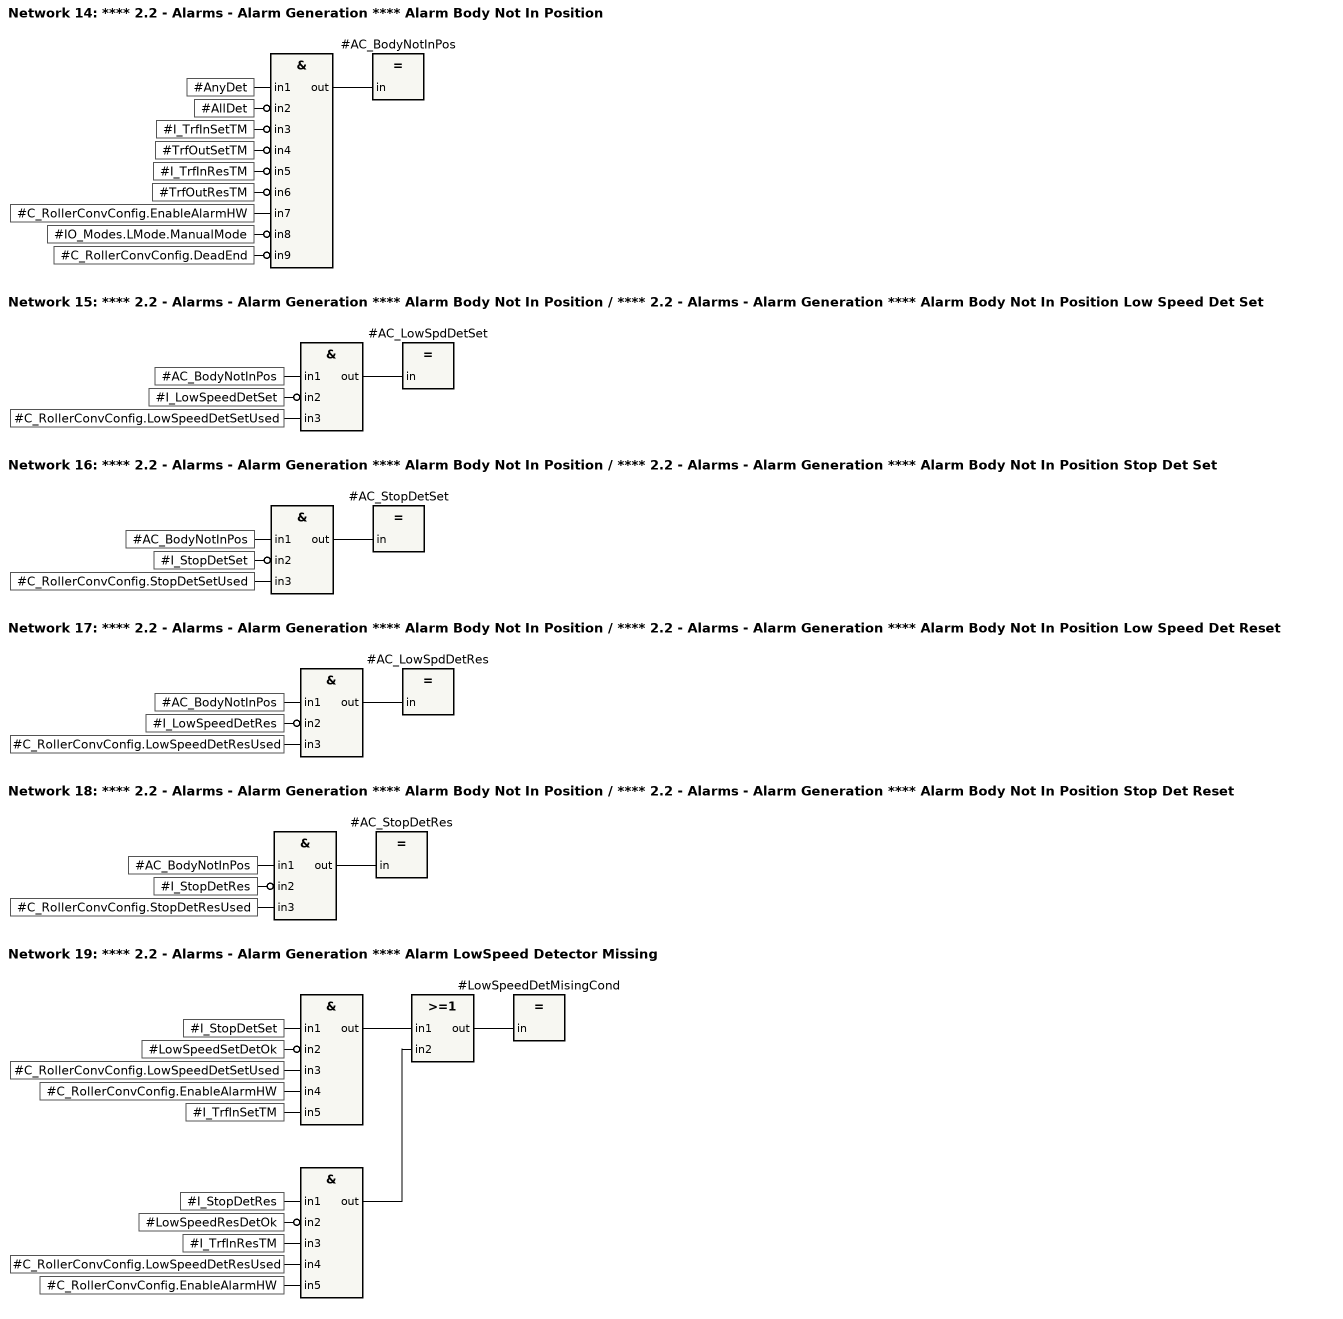
   #AC_BodyNotInPos := #AnyDet AND NOT #AllDet AND NOT #I_TrfInSetTM AND NOT #TrfOutSetTM AND NOT #I_TrfInResTM AND NOT #TrfOutResTM AND #C_RollerConvConfig.EnableAlarmHW AND NOT #IO_Modes.LMode.ManualMode AND NOT #C_RollerConvConfig.DeadEnd;
END_REGION

REGION Network 15: **** 2.2 - Alarms - Alarm Generation **** Alarm Body Not In Position / **** 2.2 - Alarms - Alarm Generation **** Alarm Body Not In Position Low Speed Det Set
   // Alarm Body Not In Position / Alarm Body Not In Position Low Speed Det Set
   #AC_LowSpdDetSet := #AC_BodyNotInPos AND NOT #I_LowSpeedDetSet AND #C_RollerConvConfig.LowSpeedDetSetUsed;
END_REGION

REGION Network 16: **** 2.2 - Alarms - Alarm Generation **** Alarm Body Not In Position / **** 2.2 - Alarms - Alarm Generation **** Alarm Body Not In Position Stop Det Set
   // Alarm Body Not In Position / Alarm Body Not In Position Stop Det Set
   #AC_StopDetSet := #AC_BodyNotInPos AND NOT #I_StopDetSet AND #C_RollerConvConfig.StopDetSetUsed;
END_REGION

REGION Network 17: **** 2.2 - Alarms - Alarm Generation **** Alarm Body Not In Position / **** 2.2 - Alarms - Alarm Generation **** Alarm Body Not In Position Low Speed Det Reset
   // Alarm Body Not In Position / Alarm Body Not In Position Low Speed Det Reset
   #AC_LowSpdDetRes := #AC_BodyNotInPos AND NOT #I_LowSpeedDetRes AND #C_RollerConvConfig.LowSpeedDetResUsed;
END_REGION

REGION Network 18: **** 2.2 - Alarms - Alarm Generation **** Alarm Body Not In Position / **** 2.2 - Alarms - Alarm Generation **** Alarm Body Not In Position Stop Det Reset
   // Alarm Body Not In Position / Alarm Body Not In Position Stop Det Reset
   #AC_StopDetRes := #AC_BodyNotInPos AND NOT #I_StopDetRes AND #C_RollerConvConfig.StopDetResUsed;
END_REGION

REGION Network 19: **** 2.2 - Alarms - Alarm Generation **** Alarm LowSpeed Detector Missing
   // Alarm LowSpeed Detector Missing
   #LowSpeedDetMisingCond := (#I_StopDetSet AND NOT #LowSpeedSetDetOk AND #C_RollerConvConfig.LowSpeedDetSetUsed AND #C_RollerConvConfig.EnableAlarmHW AND #I_TrfInSetTM) OR (#I_StopDetRes AND NOT #LowSpeedResDetOk AND #I_TrfInResTM AND #C_RollerConvConfig.LowSpeedDetResUsed AND #C_RollerConvConfig.EnableAlarmHW);
END_REGION

REGION Network 20: **** 2.2 - Alarms - Alarm Generation **** Alarm LowSpeed Detector Missing
   // Alarm LowSpeed Detector Missing
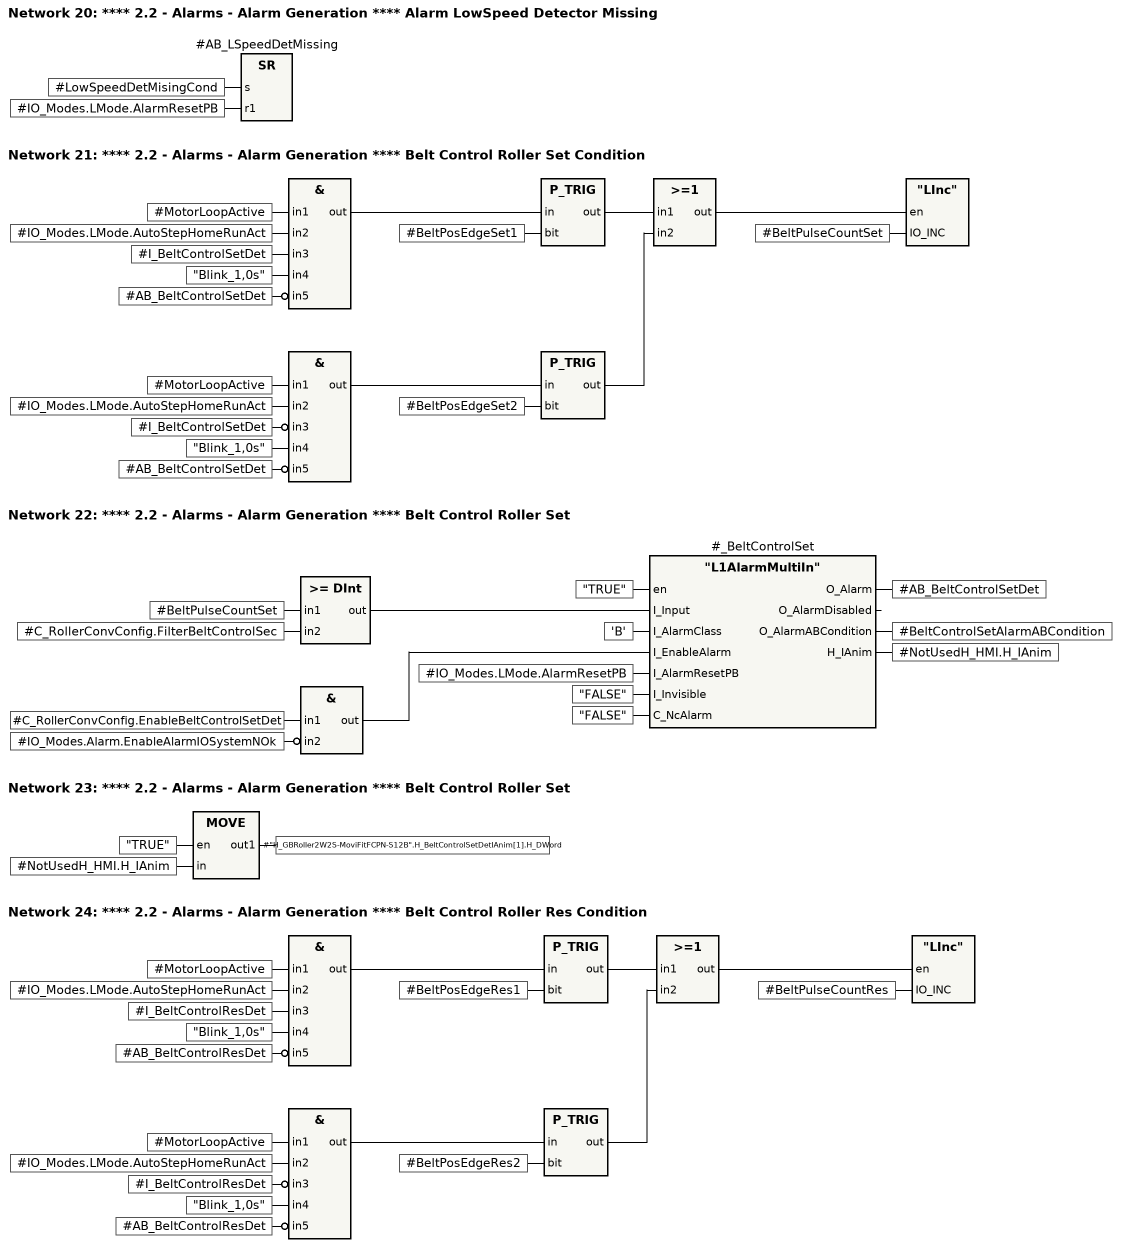
   IF #LowSpeedDetMisingCond THEN
       #AB_LSpeedDetMissing := TRUE;   // SR flip-flop
   END_IF;
   IF #IO_Modes.LMode.AlarmResetPB THEN #AB_LSpeedDetMissing := FALSE; END_IF;
END_REGION

REGION Network 21: **** 2.2 - Alarms - Alarm Generation **** Belt Control Roller Set Condition
   // Belt Control Roller Set Condition
   #_w1 := #MotorLoopActive AND #IO_Modes.LMode.AutoStepHomeRunAct AND #I_BeltControlSetDet AND "Blink_1,0s" AND NOT #AB_BeltControlSetDet;
   #_w2 := #_w1 AND NOT #BeltPosEdgeSet1;   // rising edge
   #BeltPosEdgeSet1 := #_w1;
   #_w3 := #MotorLoopActive AND #IO_Modes.LMode.AutoStepHomeRunAct AND NOT #I_BeltControlSetDet AND "Blink_1,0s" AND NOT #AB_BeltControlSetDet;
   #_w4 := #_w3 AND NOT #BeltPosEdgeSet2;   // rising edge
   #BeltPosEdgeSet2 := #_w3;
   IF #_w2 OR #_w4 THEN "LInc"(IO_INC := #BeltPulseCountSet); END_IF;
END_REGION

REGION Network 22: **** 2.2 - Alarms - Alarm Generation **** Belt Control Roller Set
   // Belt Control Roller Set
   IF "TRUE" THEN
       #_BeltControlSet(I_Input := #BeltPulseCountSet >= #C_RollerConvConfig.FilterBeltControlSec,   // "L1AlarmMultiIn"
                        I_AlarmClass := 'B',
                        I_EnableAlarm := #C_RollerConvConfig.EnableBeltControlSetDet AND NOT #IO_Modes.Alarm.EnableAlarmIOSystemNOk,
                        I_AlarmResetPB := #IO_Modes.LMode.AlarmResetPB,
                        I_Invisible := "FALSE",
                        C_NcAlarm := "FALSE",
                        O_Alarm => #AB_BeltControlSetDet,
                        O_AlarmABCondition => #BeltControlSetAlarmABCondition,
                        H_IAnim => #NotUsedH_HMI.H_IAnim);
   END_IF;
END_REGION

REGION Network 23: **** 2.2 - Alarms - Alarm Generation **** Belt Control Roller Set
   // Belt Control Roller Set
   IF "TRUE" THEN
       #"H_GBRoller2W2S-MoviFitFCPN-S12B".H_BeltControlSetDetIAnim[1].H_DWord := #NotUsedH_HMI.H_IAnim;
   END_IF;
END_REGION

REGION Network 24: **** 2.2 - Alarms - Alarm Generation **** Belt Control Roller Res Condition
   // Belt Control Roller Set Condition
   #_w1 := #MotorLoopActive AND #IO_Modes.LMode.AutoStepHomeRunAct AND #I_BeltControlResDet AND "Blink_1,0s" AND NOT #AB_BeltControlResDet;
   #_w2 := #_w1 AND NOT #BeltPosEdgeRes1;   // rising edge
   #BeltPosEdgeRes1 := #_w1;
   #_w3 := #MotorLoopActive AND #IO_Modes.LMode.AutoStepHomeRunAct AND NOT #I_BeltControlResDet AND "Blink_1,0s" AND NOT #AB_BeltControlResDet;
   #_w4 := #_w3 AND NOT #BeltPosEdgeRes2;   // rising edge
   #BeltPosEdgeRes2 := #_w3;
   IF #_w2 OR #_w4 THEN "LInc"(IO_INC := #BeltPulseCountRes); END_IF;
END_REGION

REGION Network 25: **** 2.2 - Alarms - Alarm Generation **** Belt Control Roller Res
   // Belt Control Roller Res
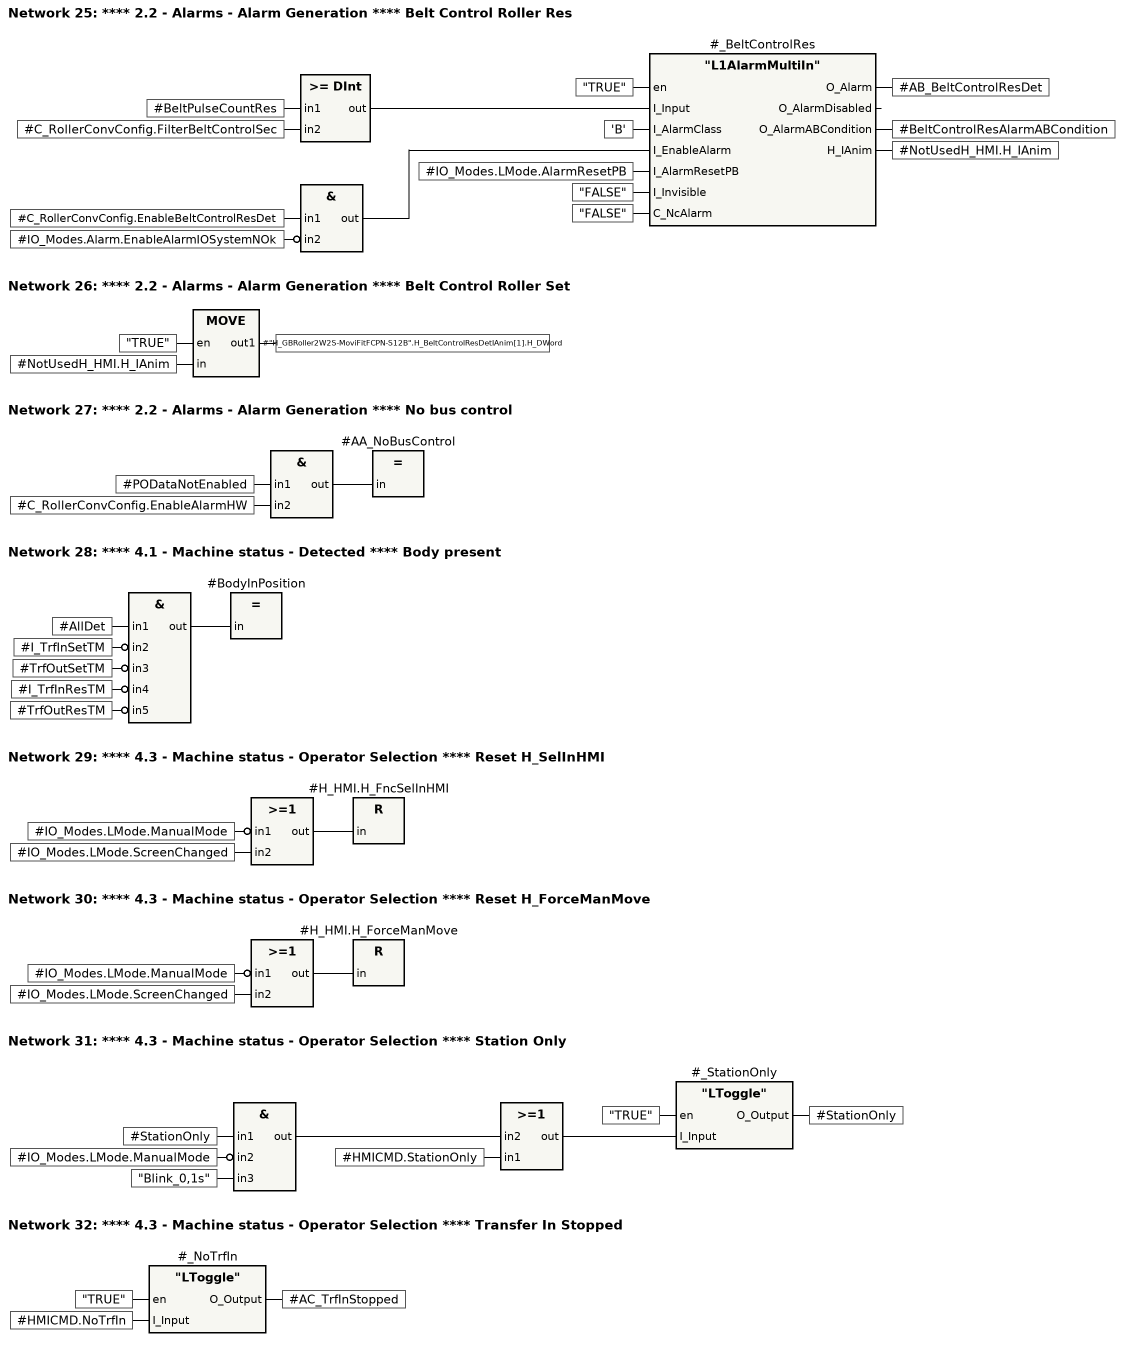
   IF "TRUE" THEN
       #_BeltControlRes(I_Input := #BeltPulseCountRes >= #C_RollerConvConfig.FilterBeltControlSec,   // "L1AlarmMultiIn"
                        I_AlarmClass := 'B',
                        I_EnableAlarm := #C_RollerConvConfig.EnableBeltControlResDet AND NOT #IO_Modes.Alarm.EnableAlarmIOSystemNOk,
                        I_AlarmResetPB := #IO_Modes.LMode.AlarmResetPB,
                        I_Invisible := "FALSE",
                        C_NcAlarm := "FALSE",
                        O_Alarm => #AB_BeltControlResDet,
                        O_AlarmABCondition => #BeltControlResAlarmABCondition,
                        H_IAnim => #NotUsedH_HMI.H_IAnim);
   END_IF;
END_REGION

REGION Network 26: **** 2.2 - Alarms - Alarm Generation **** Belt Control Roller Set
   // Belt Control Roller Set
   IF "TRUE" THEN
       #"H_GBRoller2W2S-MoviFitFCPN-S12B".H_BeltControlResDetIAnim[1].H_DWord := #NotUsedH_HMI.H_IAnim;
   END_IF;
END_REGION

REGION Network 27: **** 2.2 - Alarms - Alarm Generation **** No bus control
   #AA_NoBusControl := #PODataNotEnabled AND #C_RollerConvConfig.EnableAlarmHW;
END_REGION

REGION Network 28: **** 4.1 - Machine status - Detected **** Body present
   // Body present
   #BodyInPosition := #AllDet AND NOT #I_TrfInSetTM AND NOT #TrfOutSetTM AND NOT #I_TrfInResTM AND NOT #TrfOutResTM;
END_REGION

REGION Network 29: **** 4.3 - Machine status - Operator Selection **** Reset H_SelInHMI
   // Reset H_SelInHMI
   IF NOT #IO_Modes.LMode.ManualMode OR #IO_Modes.LMode.ScreenChanged THEN
       #H_HMI.H_FncSelInHMI := FALSE;
   END_IF;
END_REGION

REGION Network 30: **** 4.3 - Machine status - Operator Selection **** Reset H_ForceManMove
   // Reset H_ForceManMove
   IF NOT #IO_Modes.LMode.ManualMode OR #IO_Modes.LMode.ScreenChanged THEN
       #H_HMI.H_ForceManMove := FALSE;
   END_IF;
END_REGION

REGION Network 31: **** 4.3 - Machine status - Operator Selection **** Station Only
   // Reset H_ForceManMove
   IF "TRUE" THEN
       #_StationOnly(I_Input := (#StationOnly AND NOT #IO_Modes.LMode.ManualMode AND "Blink_0,1s") OR #HMICMD.StationOnly,   // "LToggle"
                     O_Output => #StationOnly);
   END_IF;
END_REGION

REGION Network 32: **** 4.3 - Machine status - Operator Selection **** Transfer In Stopped
   // Transfer In Stopped
   IF "TRUE" THEN
       #_NoTrfIn(I_Input := #HMICMD.NoTrfIn, O_Output => #AC_TrfInStopped);   // "LToggle"
   END_IF;
END_REGION

REGION Network 33: **** 4.6 - Machine status - Indications **** Transfer memory set
   // Transfer memory set
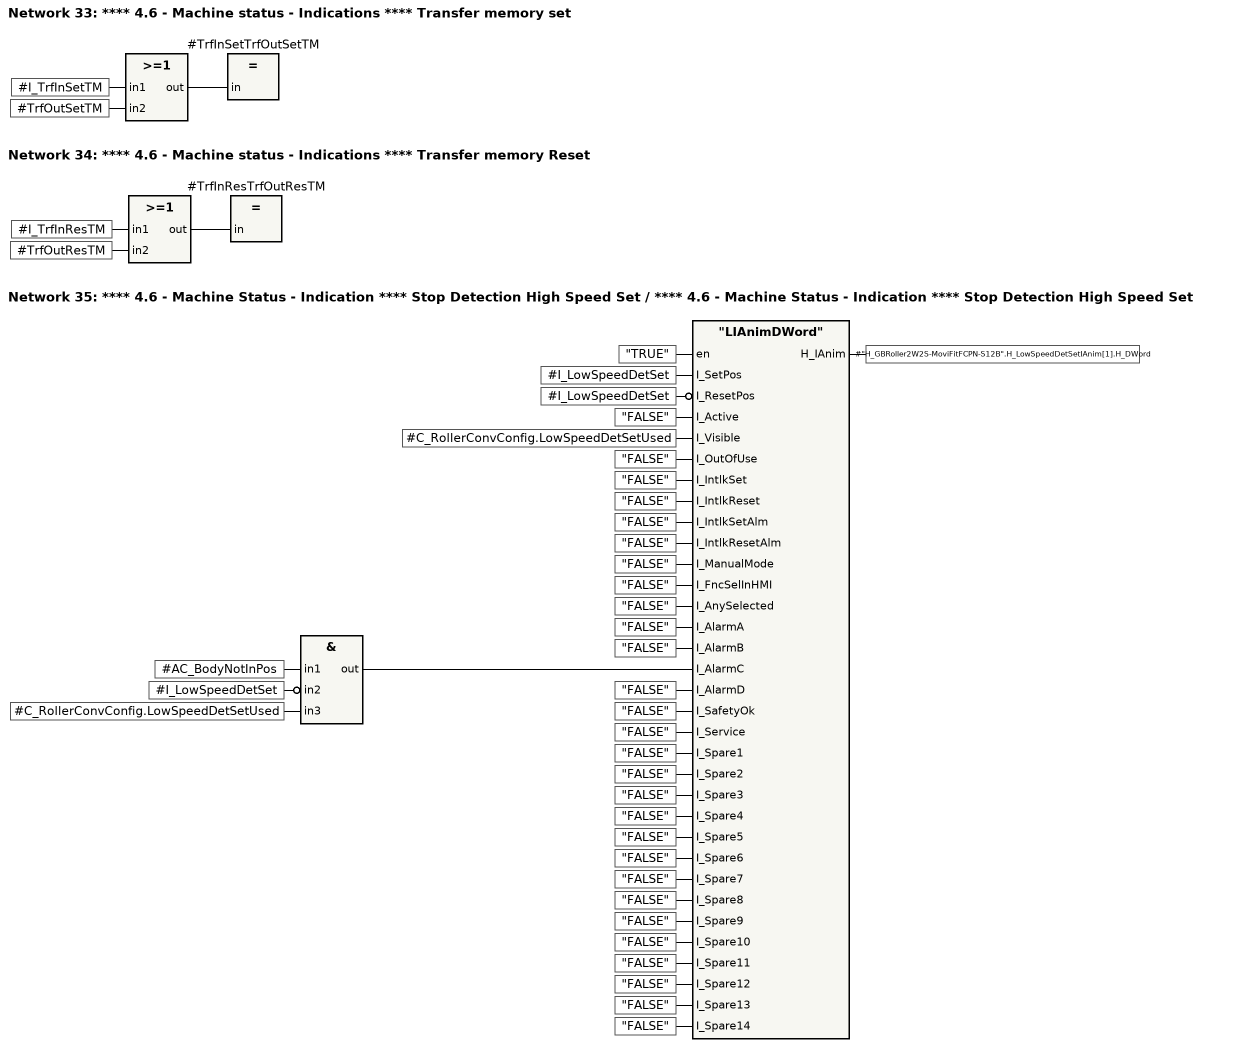
   #TrfInSetTrfOutSetTM := #I_TrfInSetTM OR #TrfOutSetTM;
END_REGION

REGION Network 34: **** 4.6 - Machine status - Indications **** Transfer memory Reset
   // Transfer memory Reset
   #TrfInResTrfOutResTM := #I_TrfInResTM OR #TrfOutResTM;
END_REGION

REGION Network 35: **** 4.6 - Machine Status - Indication **** Stop Detection High Speed Set / **** 4.6 - Machine Status - Indication **** Stop Detection High Speed Set
   // Stop Detection High Speed Set
   IF "TRUE" THEN
       "LIAnimDWord"(I_SetPos := #I_LowSpeedDetSet,
                     I_ResetPos := NOT #I_LowSpeedDetSet,
                     I_Active := "FALSE",
                     I_Visible := #C_RollerConvConfig.LowSpeedDetSetUsed,
                     I_OutOfUse := "FALSE",
                     I_IntlkSet := "FALSE",
                     I_IntlkReset := "FALSE",
                     I_IntlkSetAlm := "FALSE",
                     I_IntlkResetAlm := "FALSE",
                     I_ManualMode := "FALSE",
                     I_FncSelInHMI := "FALSE",
                     I_AnySelected := "FALSE",
                     I_AlarmA := "FALSE",
                     I_AlarmB := "FALSE",
                     I_AlarmC := #AC_BodyNotInPos AND NOT #I_LowSpeedDetSet AND #C_RollerConvConfig.LowSpeedDetSetUsed,
                     I_AlarmD := "FALSE",
                     I_SafetyOk := "FALSE",
                     I_Service := "FALSE",
                     I_Spare1 := "FALSE",
                     I_Spare2 := "FALSE",
                     I_Spare3 := "FALSE",
                     I_Spare4 := "FALSE",
                     I_Spare5 := "FALSE",
                     I_Spare6 := "FALSE",
                     I_Spare7 := "FALSE",
                     I_Spare8 := "FALSE",
                     I_Spare9 := "FALSE",
                     I_Spare10 := "FALSE",
                     I_Spare11 := "FALSE",
                     I_Spare12 := "FALSE",
                     I_Spare13 := "FALSE",
                     I_Spare14 := "FALSE",
                     H_IAnim => #"H_GBRoller2W2S-MoviFitFCPN-S12B".H_LowSpeedDetSetIAnim[1].H_DWord);
   END_IF;
END_REGION

REGION Network 36: **** 4.6 - Machine Status - Indication **** Stop Detection set
   // Stop detection set
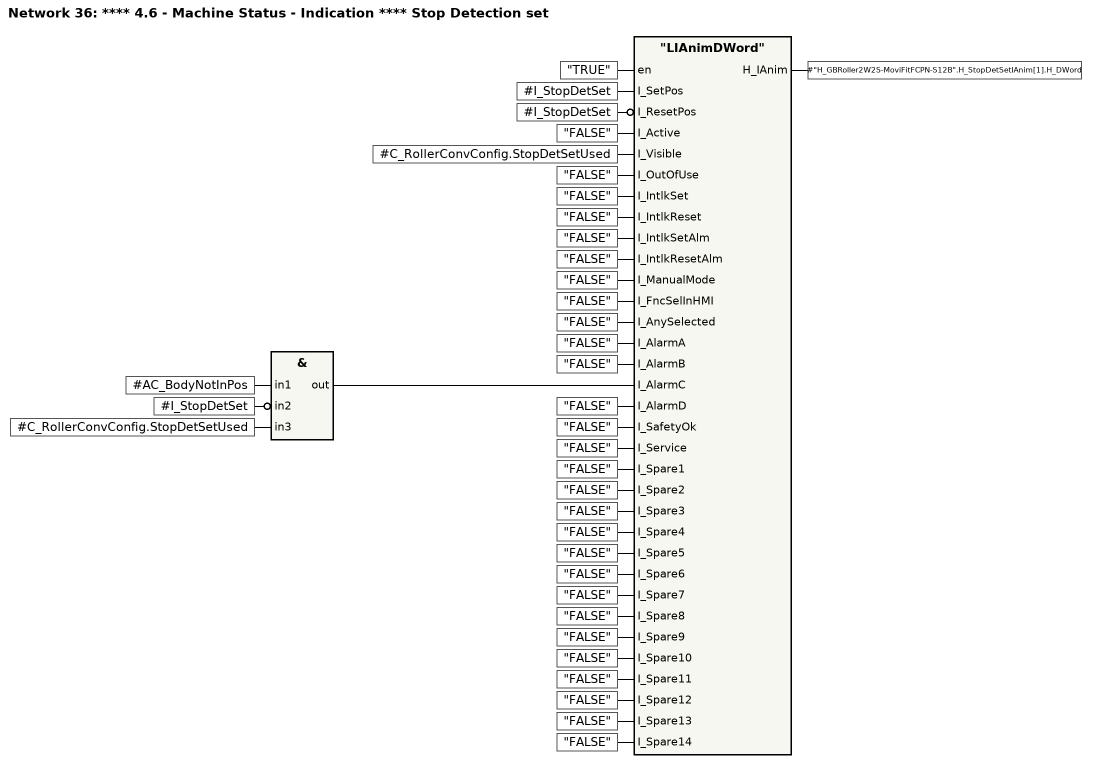
   IF "TRUE" THEN
       "LIAnimDWord"(I_SetPos := #I_StopDetSet,
                     I_ResetPos := NOT #I_StopDetSet,
                     I_Active := "FALSE",
                     I_Visible := #C_RollerConvConfig.StopDetSetUsed,
                     I_OutOfUse := "FALSE",
                     I_IntlkSet := "FALSE",
                     I_IntlkReset := "FALSE",
                     I_IntlkSetAlm := "FALSE",
                     I_IntlkResetAlm := "FALSE",
                     I_ManualMode := "FALSE",
                     I_FncSelInHMI := "FALSE",
                     I_AnySelected := "FALSE",
                     I_AlarmA := "FALSE",
                     I_AlarmB := "FALSE",
                     I_AlarmC := #AC_BodyNotInPos AND NOT #I_StopDetSet AND #C_RollerConvConfig.StopDetSetUsed,
                     I_AlarmD := "FALSE",
                     I_SafetyOk := "FALSE",
                     I_Service := "FALSE",
                     I_Spare1 := "FALSE",
                     I_Spare2 := "FALSE",
                     I_Spare3 := "FALSE",
                     I_Spare4 := "FALSE",
                     I_Spare5 := "FALSE",
                     I_Spare6 := "FALSE",
                     I_Spare7 := "FALSE",
                     I_Spare8 := "FALSE",
                     I_Spare9 := "FALSE",
                     I_Spare10 := "FALSE",
                     I_Spare11 := "FALSE",
                     I_Spare12 := "FALSE",
                     I_Spare13 := "FALSE",
                     I_Spare14 := "FALSE",
                     H_IAnim => #"H_GBRoller2W2S-MoviFitFCPN-S12B".H_StopDetSetIAnim[1].H_DWord);
   END_IF;
END_REGION

REGION Network 37: **** 4.6 - Machine Status - Indication **** Stop Detection High Speed Reset
   // Stop detection High Speed Reset
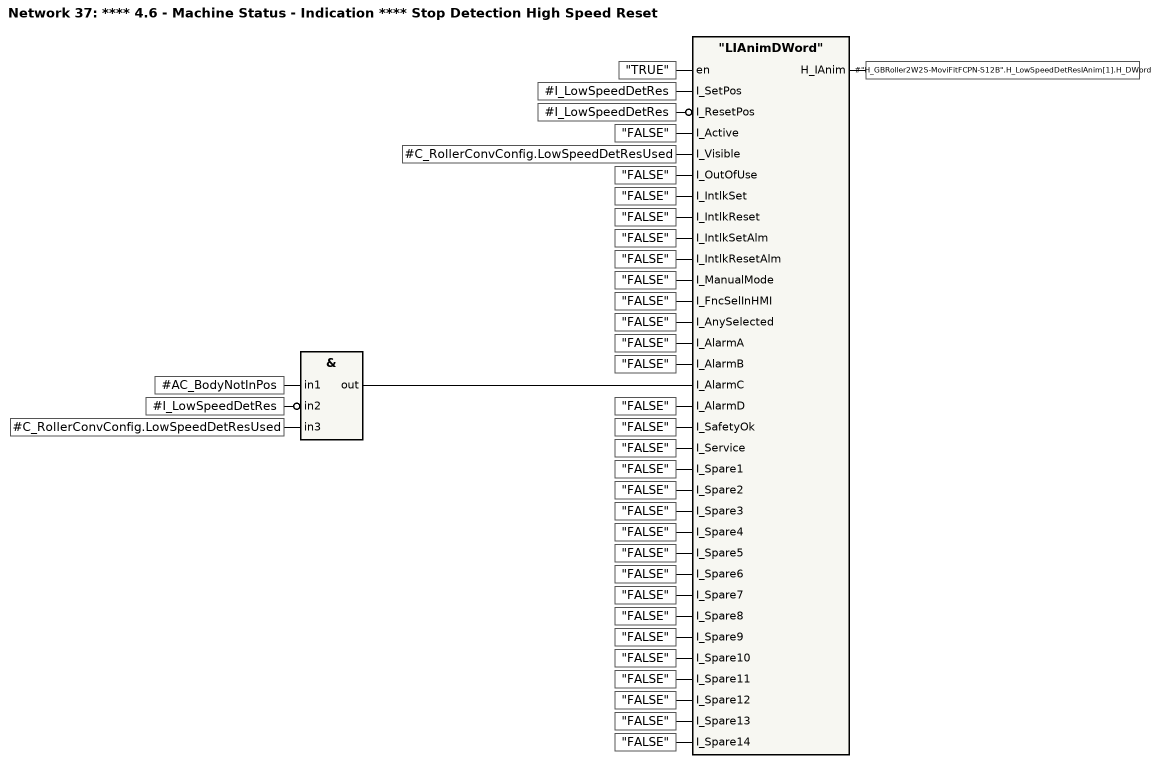
   IF "TRUE" THEN
       "LIAnimDWord"(I_SetPos := #I_LowSpeedDetRes,
                     I_ResetPos := NOT #I_LowSpeedDetRes,
                     I_Active := "FALSE",
                     I_Visible := #C_RollerConvConfig.LowSpeedDetResUsed,
                     I_OutOfUse := "FALSE",
                     I_IntlkSet := "FALSE",
                     I_IntlkReset := "FALSE",
                     I_IntlkSetAlm := "FALSE",
                     I_IntlkResetAlm := "FALSE",
                     I_ManualMode := "FALSE",
                     I_FncSelInHMI := "FALSE",
                     I_AnySelected := "FALSE",
                     I_AlarmA := "FALSE",
                     I_AlarmB := "FALSE",
                     I_AlarmC := #AC_BodyNotInPos AND NOT #I_LowSpeedDetRes AND #C_RollerConvConfig.LowSpeedDetResUsed,
                     I_AlarmD := "FALSE",
                     I_SafetyOk := "FALSE",
                     I_Service := "FALSE",
                     I_Spare1 := "FALSE",
                     I_Spare2 := "FALSE",
                     I_Spare3 := "FALSE",
                     I_Spare4 := "FALSE",
                     I_Spare5 := "FALSE",
                     I_Spare6 := "FALSE",
                     I_Spare7 := "FALSE",
                     I_Spare8 := "FALSE",
                     I_Spare9 := "FALSE",
                     I_Spare10 := "FALSE",
                     I_Spare11 := "FALSE",
                     I_Spare12 := "FALSE",
                     I_Spare13 := "FALSE",
                     I_Spare14 := "FALSE",
                     H_IAnim => #"H_GBRoller2W2S-MoviFitFCPN-S12B".H_LowSpeedDetResIAnim[1].H_DWord);
   END_IF;
END_REGION

REGION Network 38: **** 4.6 - Machine Status - Indication **** Stop Detection Reset
   // Stop detection Reset
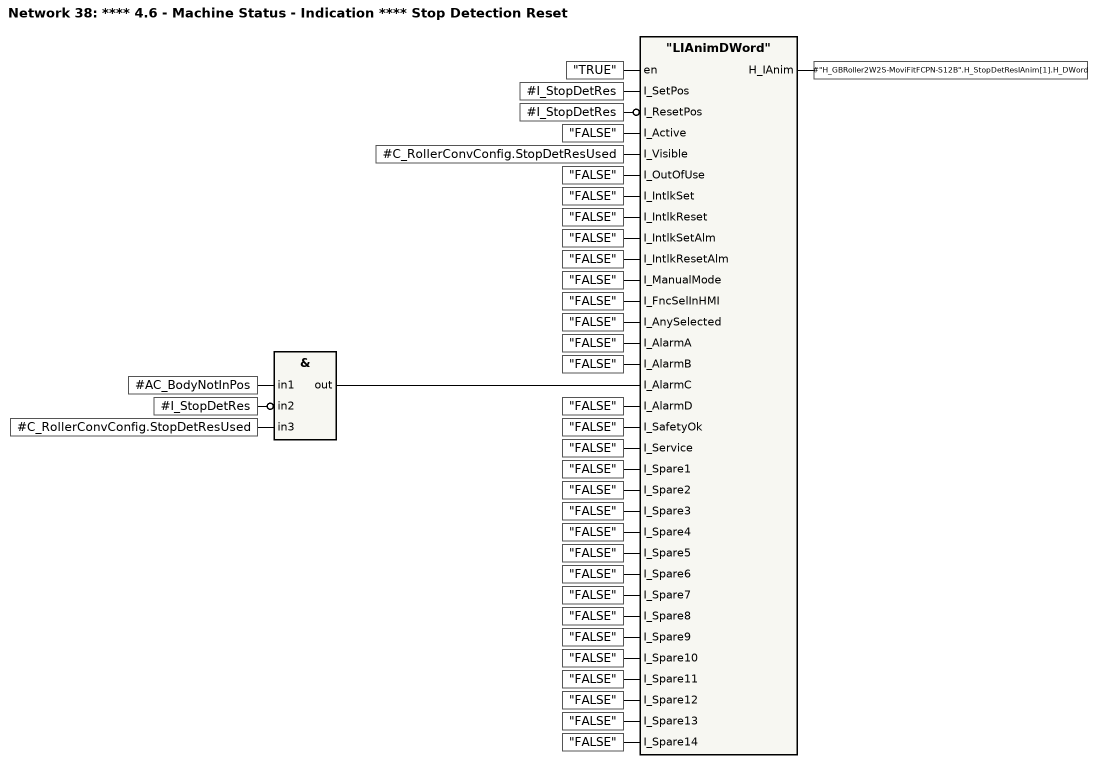
   IF "TRUE" THEN
       "LIAnimDWord"(I_SetPos := #I_StopDetRes,
                     I_ResetPos := NOT #I_StopDetRes,
                     I_Active := "FALSE",
                     I_Visible := #C_RollerConvConfig.StopDetResUsed,
                     I_OutOfUse := "FALSE",
                     I_IntlkSet := "FALSE",
                     I_IntlkReset := "FALSE",
                     I_IntlkSetAlm := "FALSE",
                     I_IntlkResetAlm := "FALSE",
                     I_ManualMode := "FALSE",
                     I_FncSelInHMI := "FALSE",
                     I_AnySelected := "FALSE",
                     I_AlarmA := "FALSE",
                     I_AlarmB := "FALSE",
                     I_AlarmC := #AC_BodyNotInPos AND NOT #I_StopDetRes AND #C_RollerConvConfig.StopDetResUsed,
                     I_AlarmD := "FALSE",
                     I_SafetyOk := "FALSE",
                     I_Service := "FALSE",
                     I_Spare1 := "FALSE",
                     I_Spare2 := "FALSE",
                     I_Spare3 := "FALSE",
                     I_Spare4 := "FALSE",
                     I_Spare5 := "FALSE",
                     I_Spare6 := "FALSE",
                     I_Spare7 := "FALSE",
                     I_Spare8 := "FALSE",
                     I_Spare9 := "FALSE",
                     I_Spare10 := "FALSE",
                     I_Spare11 := "FALSE",
                     I_Spare12 := "FALSE",
                     I_Spare13 := "FALSE",
                     I_Spare14 := "FALSE",
                     H_IAnim => #"H_GBRoller2W2S-MoviFitFCPN-S12B".H_StopDetResIAnim[1].H_DWord);
   END_IF;
END_REGION

REGION Network 39: **** 4.6 - Machine Status - Indication **** Stop Detection Reset / **** 4.6 - Machine Status - Indication **** Occupied Detection
   // Stop detection Reset / Occupied Detection
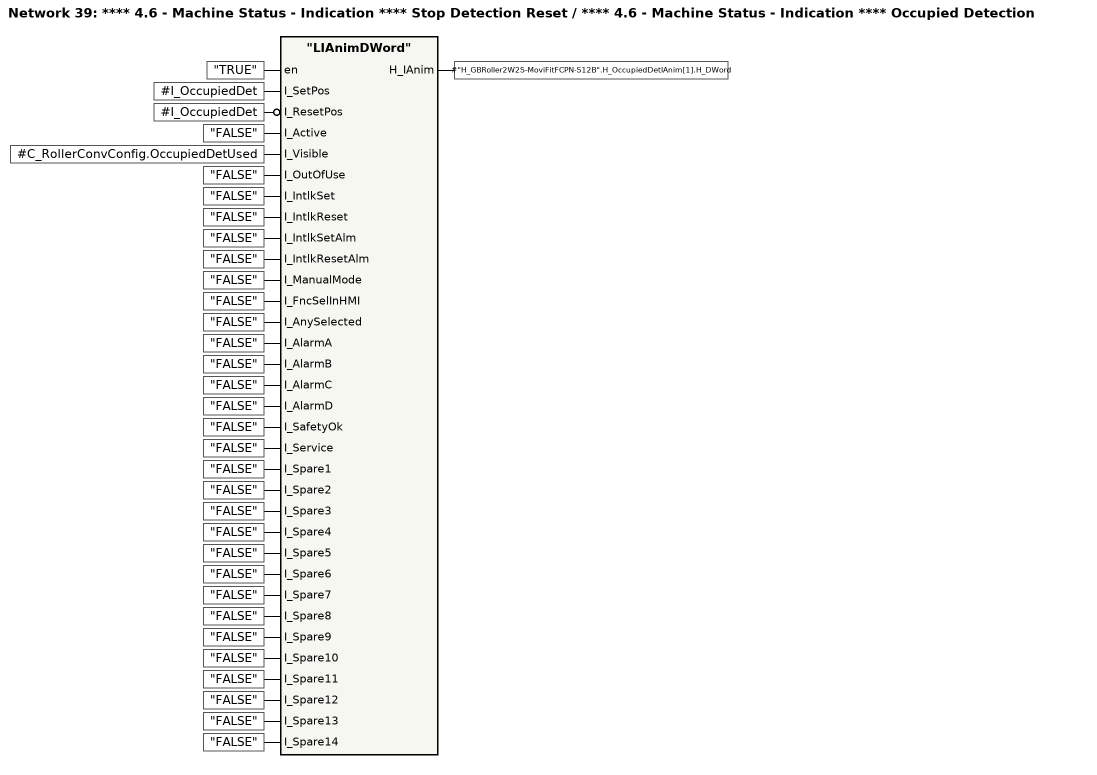
   IF "TRUE" THEN
       "LIAnimDWord"(I_SetPos := #I_OccupiedDet,
                     I_ResetPos := NOT #I_OccupiedDet,
                     I_Active := "FALSE",
                     I_Visible := #C_RollerConvConfig.OccupiedDetUsed,
                     I_OutOfUse := "FALSE",
                     I_IntlkSet := "FALSE",
                     I_IntlkReset := "FALSE",
                     I_IntlkSetAlm := "FALSE",
                     I_IntlkResetAlm := "FALSE",
                     I_ManualMode := "FALSE",
                     I_FncSelInHMI := "FALSE",
                     I_AnySelected := "FALSE",
                     I_AlarmA := "FALSE",
                     I_AlarmB := "FALSE",
                     I_AlarmC := "FALSE",
                     I_AlarmD := "FALSE",
                     I_SafetyOk := "FALSE",
                     I_Service := "FALSE",
                     I_Spare1 := "FALSE",
                     I_Spare2 := "FALSE",
                     I_Spare3 := "FALSE",
                     I_Spare4 := "FALSE",
                     I_Spare5 := "FALSE",
                     I_Spare6 := "FALSE",
                     I_Spare7 := "FALSE",
                     I_Spare8 := "FALSE",
                     I_Spare9 := "FALSE",
                     I_Spare10 := "FALSE",
                     I_Spare11 := "FALSE",
                     I_Spare12 := "FALSE",
                     I_Spare13 := "FALSE",
                     I_Spare14 := "FALSE",
                     H_IAnim => #"H_GBRoller2W2S-MoviFitFCPN-S12B".H_OccupiedDetIAnim[1].H_DWord);
   END_IF;
END_REGION

REGION Network 40: **** 4.6 - Machine Status - Indication **** Icon Animation
   // Icon Animation
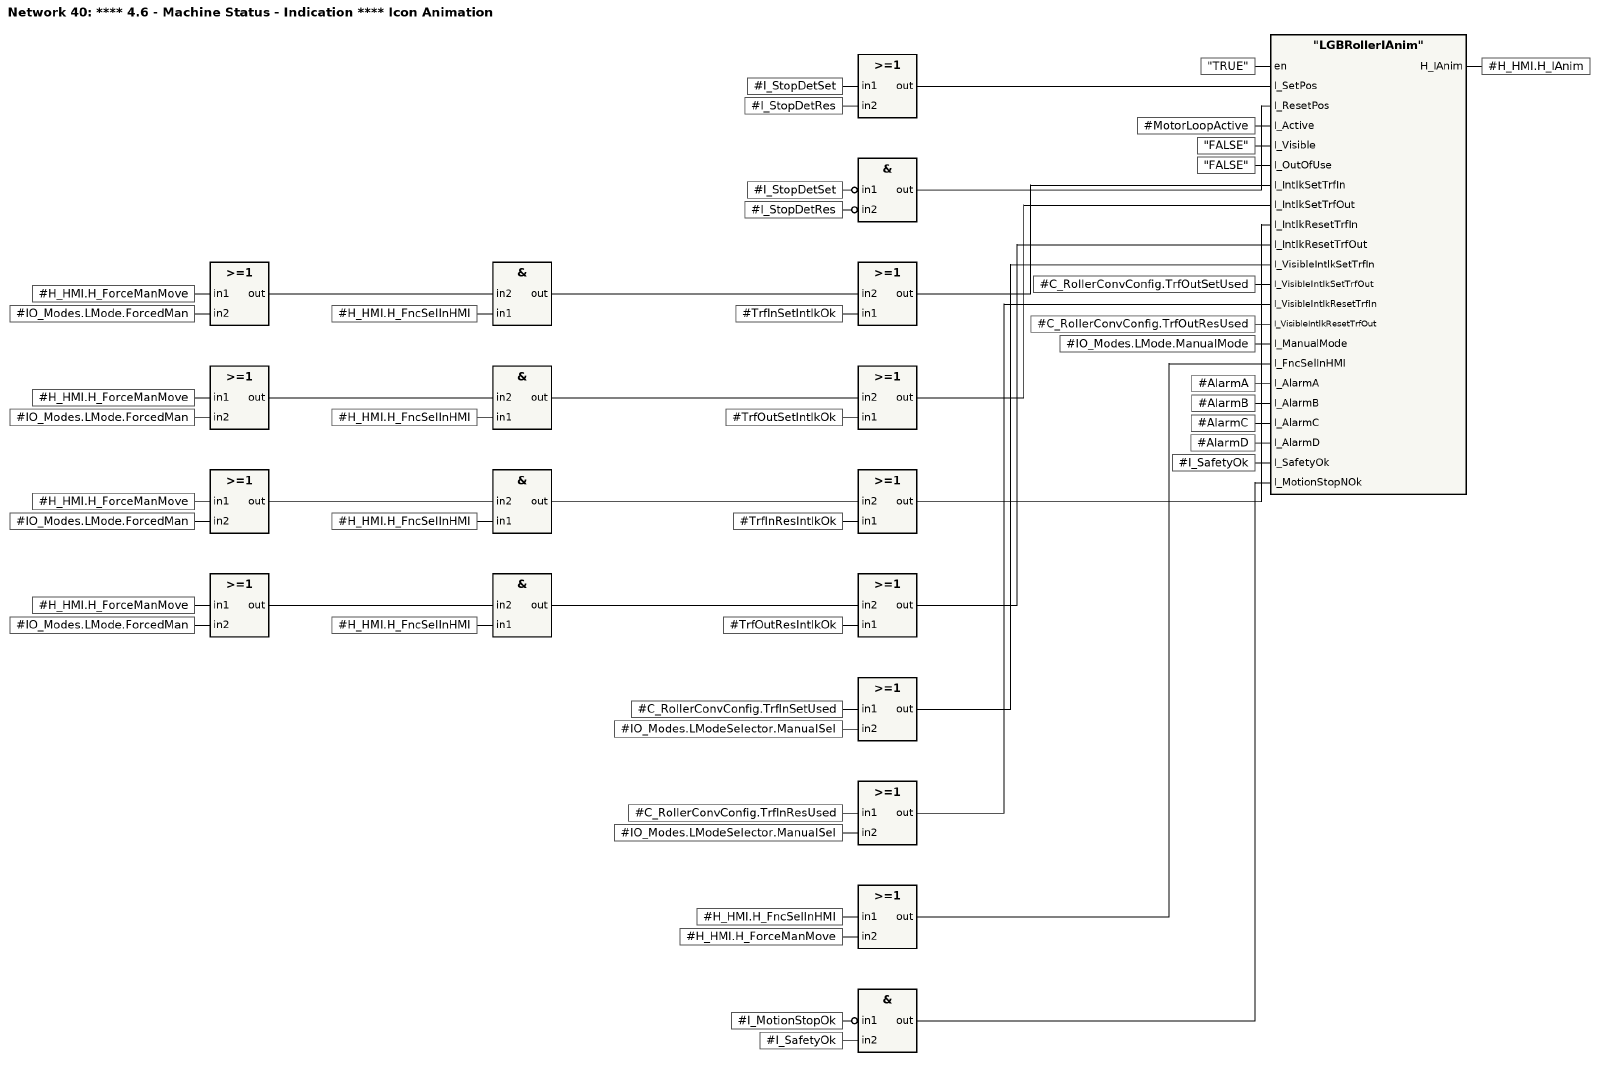
   IF "TRUE" THEN
       "LGBRollerIAnim"(I_SetPos := #I_StopDetSet OR #I_StopDetRes,
                        I_ResetPos := NOT #I_StopDetSet AND NOT #I_StopDetRes,
                        I_Active := #MotorLoopActive,
                        I_Visible := "FALSE",
                        I_OutOfUse := "FALSE",
                        I_IntlkSetTrfIn := ((#H_HMI.H_ForceManMove OR #IO_Modes.LMode.ForcedMan) AND #H_HMI.H_FncSelInHMI) OR #TrfInSetIntlkOk,
                        I_IntlkSetTrfOut := ((#H_HMI.H_ForceManMove OR #IO_Modes.LMode.ForcedMan) AND #H_HMI.H_FncSelInHMI) OR #TrfOutSetIntlkOk,
                        I_IntlkResetTrfIn := ((#H_HMI.H_ForceManMove OR #IO_Modes.LMode.ForcedMan) AND #H_HMI.H_FncSelInHMI) OR #TrfInResIntlkOk,
                        I_IntlkResetTrfOut := ((#H_HMI.H_ForceManMove OR #IO_Modes.LMode.ForcedMan) AND #H_HMI.H_FncSelInHMI) OR #TrfOutResIntlkOk,
                        I_VisibleIntlkSetTrfIn := #C_RollerConvConfig.TrfInSetUsed OR #IO_Modes.LModeSelector.ManualSel,
                        I_VisibleIntlkSetTrfOut := #C_RollerConvConfig.TrfOutSetUsed,
                        I_VisibleIntlkResetTrfIn := #C_RollerConvConfig.TrfInResUsed OR #IO_Modes.LModeSelector.ManualSel,
                        I_VisibleIntlkResetTrfOut := #C_RollerConvConfig.TrfOutResUsed,
                        I_ManualMode := #IO_Modes.LMode.ManualMode,
                        I_FncSelInHMI := #H_HMI.H_FncSelInHMI OR #H_HMI.H_ForceManMove,
                        I_AlarmA := #AlarmA,
                        I_AlarmB := #AlarmB,
                        I_AlarmC := #AlarmC,
                        I_AlarmD := #AlarmD,
                        I_SafetyOk := #I_SafetyOk,
                        I_MotionStopNOk := NOT #I_MotionStopOk AND #I_SafetyOk,
                        H_IAnim => #H_HMI.H_IAnim);
   END_IF;
END_REGION

REGION Network 41: **** 4.6 - Machine Status - Indication **** Animation
   // Animation
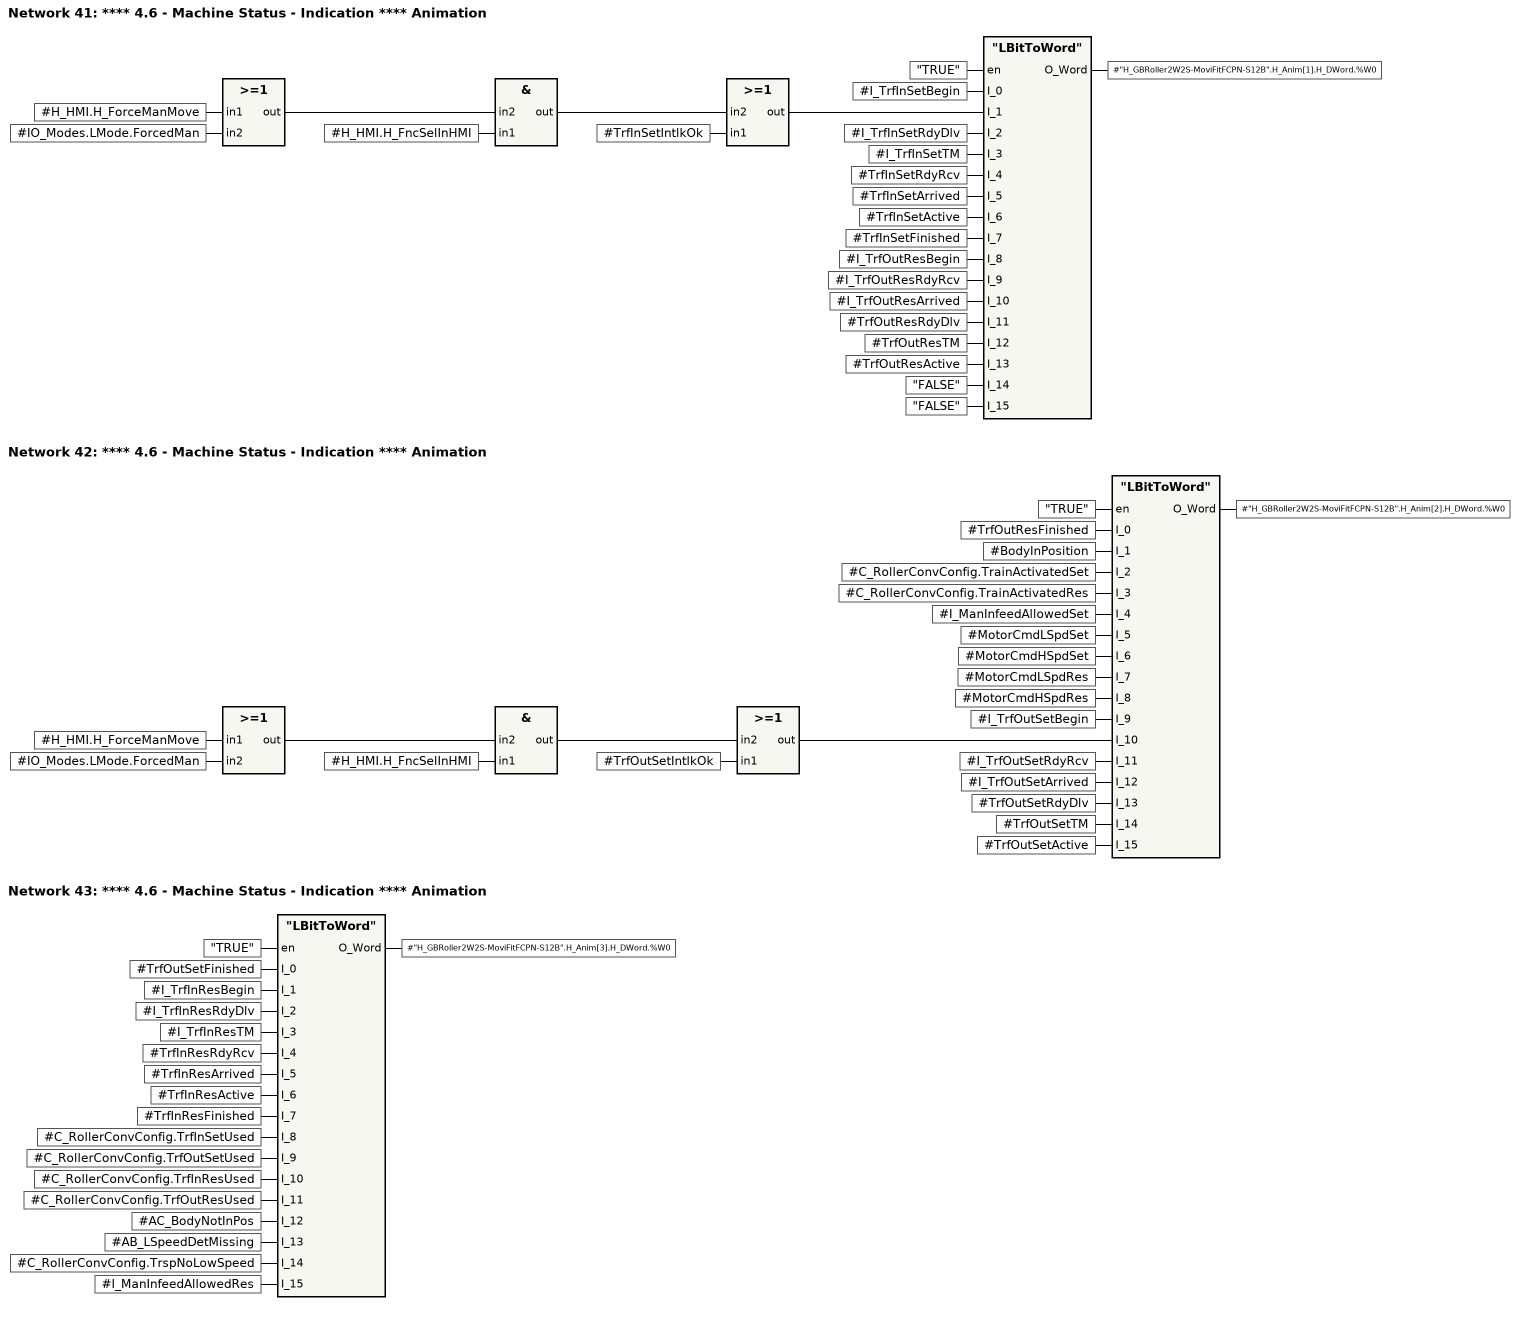
   IF "TRUE" THEN
       "LBitToWord"(I_0 := #I_TrfInSetBegin,
                    I_1 := ((#H_HMI.H_ForceManMove OR #IO_Modes.LMode.ForcedMan) AND #H_HMI.H_FncSelInHMI) OR #TrfInSetIntlkOk,
                    I_2 := #I_TrfInSetRdyDlv,
                    I_3 := #I_TrfInSetTM,
                    I_4 := #TrfInSetRdyRcv,
                    I_5 := #TrfInSetArrived,
                    I_6 := #TrfInSetActive,
                    I_7 := #TrfInSetFinished,
                    I_8 := #I_TrfOutResBegin,
                    I_9 := #I_TrfOutResRdyRcv,
                    I_10 := #I_TrfOutResArrived,
                    I_11 := #TrfOutResRdyDlv,
                    I_12 := #TrfOutResTM,
                    I_13 := #TrfOutResActive,
                    I_14 := "FALSE",
                    I_15 := "FALSE",
                    O_Word => #"H_GBRoller2W2S-MoviFitFCPN-S12B".H_Anim[1].H_DWord.%W0);
   END_IF;
END_REGION

REGION Network 42: **** 4.6 - Machine Status - Indication **** Animation
   // Animation
   IF "TRUE" THEN
       "LBitToWord"(I_0 := #TrfOutResFinished,
                    I_1 := #BodyInPosition,
                    I_2 := #C_RollerConvConfig.TrainActivatedSet,
                    I_3 := #C_RollerConvConfig.TrainActivatedRes,
                    I_4 := #I_ManInfeedAllowedSet,
                    I_5 := #MotorCmdLSpdSet,
                    I_6 := #MotorCmdHSpdSet,
                    I_7 := #MotorCmdLSpdRes,
                    I_8 := #MotorCmdHSpdRes,
                    I_9 := #I_TrfOutSetBegin,
                    I_10 := ((#H_HMI.H_ForceManMove OR #IO_Modes.LMode.ForcedMan) AND #H_HMI.H_FncSelInHMI) OR #TrfOutSetIntlkOk,
                    I_11 := #I_TrfOutSetRdyRcv,
                    I_12 := #I_TrfOutSetArrived,
                    I_13 := #TrfOutSetRdyDlv,
                    I_14 := #TrfOutSetTM,
                    I_15 := #TrfOutSetActive,
                    O_Word => #"H_GBRoller2W2S-MoviFitFCPN-S12B".H_Anim[2].H_DWord.%W0);
   END_IF;
END_REGION

REGION Network 43: **** 4.6 - Machine Status - Indication **** Animation
   // Animation
   IF "TRUE" THEN
       "LBitToWord"(I_0 := #TrfOutSetFinished,
                    I_1 := #I_TrfInResBegin,
                    I_2 := #I_TrfInResRdyDlv,
                    I_3 := #I_TrfInResTM,
                    I_4 := #TrfInResRdyRcv,
                    I_5 := #TrfInResArrived,
                    I_6 := #TrfInResActive,
                    I_7 := #TrfInResFinished,
                    I_8 := #C_RollerConvConfig.TrfInSetUsed,
                    I_9 := #C_RollerConvConfig.TrfOutSetUsed,
                    I_10 := #C_RollerConvConfig.TrfInResUsed,
                    I_11 := #C_RollerConvConfig.TrfOutResUsed,
                    I_12 := #AC_BodyNotInPos,
                    I_13 := #AB_LSpeedDetMissing,
                    I_14 := #C_RollerConvConfig.TrspNoLowSpeed,
                    I_15 := #I_ManInfeedAllowedRes,
                    O_Word => #"H_GBRoller2W2S-MoviFitFCPN-S12B".H_Anim[3].H_DWord.%W0);
   END_IF;
END_REGION

REGION Network 44: **** 4.6 - Machine Status - Indication **** Animation
   // Animation
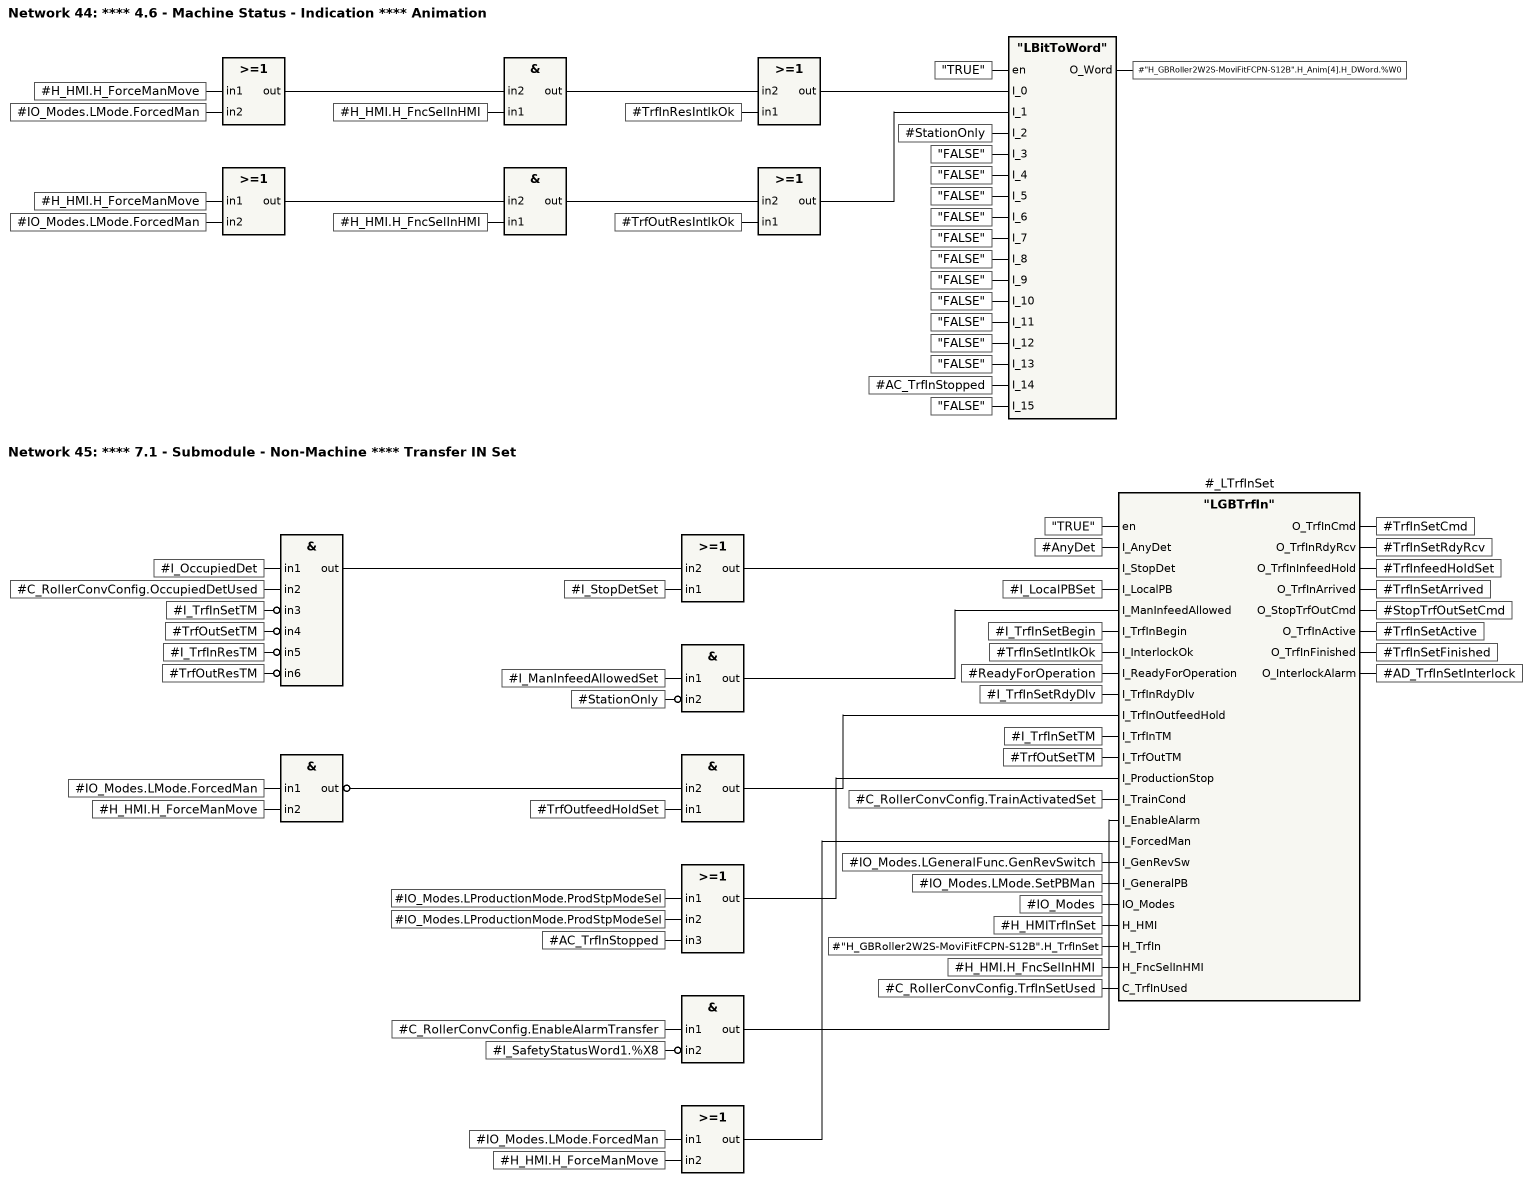
   IF "TRUE" THEN
       "LBitToWord"(I_0 := ((#H_HMI.H_ForceManMove OR #IO_Modes.LMode.ForcedMan) AND #H_HMI.H_FncSelInHMI) OR #TrfInResIntlkOk,
                    I_1 := ((#H_HMI.H_ForceManMove OR #IO_Modes.LMode.ForcedMan) AND #H_HMI.H_FncSelInHMI) OR #TrfOutResIntlkOk,
                    I_2 := #StationOnly,
                    I_3 := "FALSE",
                    I_4 := "FALSE",
                    I_5 := "FALSE",
                    I_6 := "FALSE",
                    I_7 := "FALSE",
                    I_8 := "FALSE",
                    I_9 := "FALSE",
                    I_10 := "FALSE",
                    I_11 := "FALSE",
                    I_12 := "FALSE",
                    I_13 := "FALSE",
                    I_14 := #AC_TrfInStopped,
                    I_15 := "FALSE",
                    O_Word => #"H_GBRoller2W2S-MoviFitFCPN-S12B".H_Anim[4].H_DWord.%W0);
   END_IF;
END_REGION

REGION Network 45: **** 7.1 - Submodule - Non-Machine **** Transfer IN Set
   // Transfer IN Set
   IF "TRUE" THEN
       #_LTrfInSet(I_AnyDet := #AnyDet,   // "LGBTrfIn"
                   I_StopDet := (#I_OccupiedDet AND #C_RollerConvConfig.OccupiedDetUsed AND NOT #I_TrfInSetTM AND NOT #TrfOutSetTM AND NOT #I_TrfInResTM AND NOT #TrfOutResTM) OR #I_StopDetSet,
                   I_LocalPB := #I_LocalPBSet,
                   I_ManInfeedAllowed := #I_ManInfeedAllowedSet AND NOT #StationOnly,
                   I_TrfInBegin := #I_TrfInSetBegin,
                   I_InterlockOk := #TrfInSetIntlkOk,
                   I_ReadyForOperation := #ReadyForOperation,
                   I_TrfInRdyDlv := #I_TrfInSetRdyDlv,
                   I_TrfInOutfeedHold := NOT (#IO_Modes.LMode.ForcedMan AND #H_HMI.H_ForceManMove) AND #TrfOutfeedHoldSet,
                   I_TrfInTM := #I_TrfInSetTM,
                   I_TrfOutTM := #TrfOutSetTM,
                   I_ProductionStop := #IO_Modes.LProductionMode.ProdStpModeSel OR #IO_Modes.LProductionMode.ProdStpModeSel OR #AC_TrfInStopped,
                   I_TrainCond := #C_RollerConvConfig.TrainActivatedSet,
                   I_EnableAlarm := #C_RollerConvConfig.EnableAlarmTransfer AND NOT #I_SafetyStatusWord1.%X8,
                   I_ForcedMan := #IO_Modes.LMode.ForcedMan OR #H_HMI.H_ForceManMove,
                   I_GenRevSw := #IO_Modes.LGeneralFunc.GenRevSwitch,
                   I_GeneralPB := #IO_Modes.LMode.SetPBMan,
                   IO_Modes := #IO_Modes,
                   H_HMI := #H_HMITrfInSet,
                   H_TrfIn := #"H_GBRoller2W2S-MoviFitFCPN-S12B".H_TrfInSet,
                   H_FncSelInHMI := #H_HMI.H_FncSelInHMI,
                   C_TrfInUsed := #C_RollerConvConfig.TrfInSetUsed,
                   O_TrfInCmd => #TrfInSetCmd,
                   O_TrfInRdyRcv => #TrfInSetRdyRcv,
                   O_TrfInInfeedHold => #TrfInfeedHoldSet,
                   O_TrfInArrived => #TrfInSetArrived,
                   O_StopTrfOutCmd => #StopTrfOutSetCmd,
                   O_TrfInActive => #TrfInSetActive,
                   O_TrfInFinished => #TrfInSetFinished,
                   O_InterlockAlarm => #AD_TrfInSetInterlock);
   END_IF;
END_REGION

REGION Network 46: **** 7.1 - Submodule - Non-Machine **** Transfer Out Set
   // Transfer Out Set
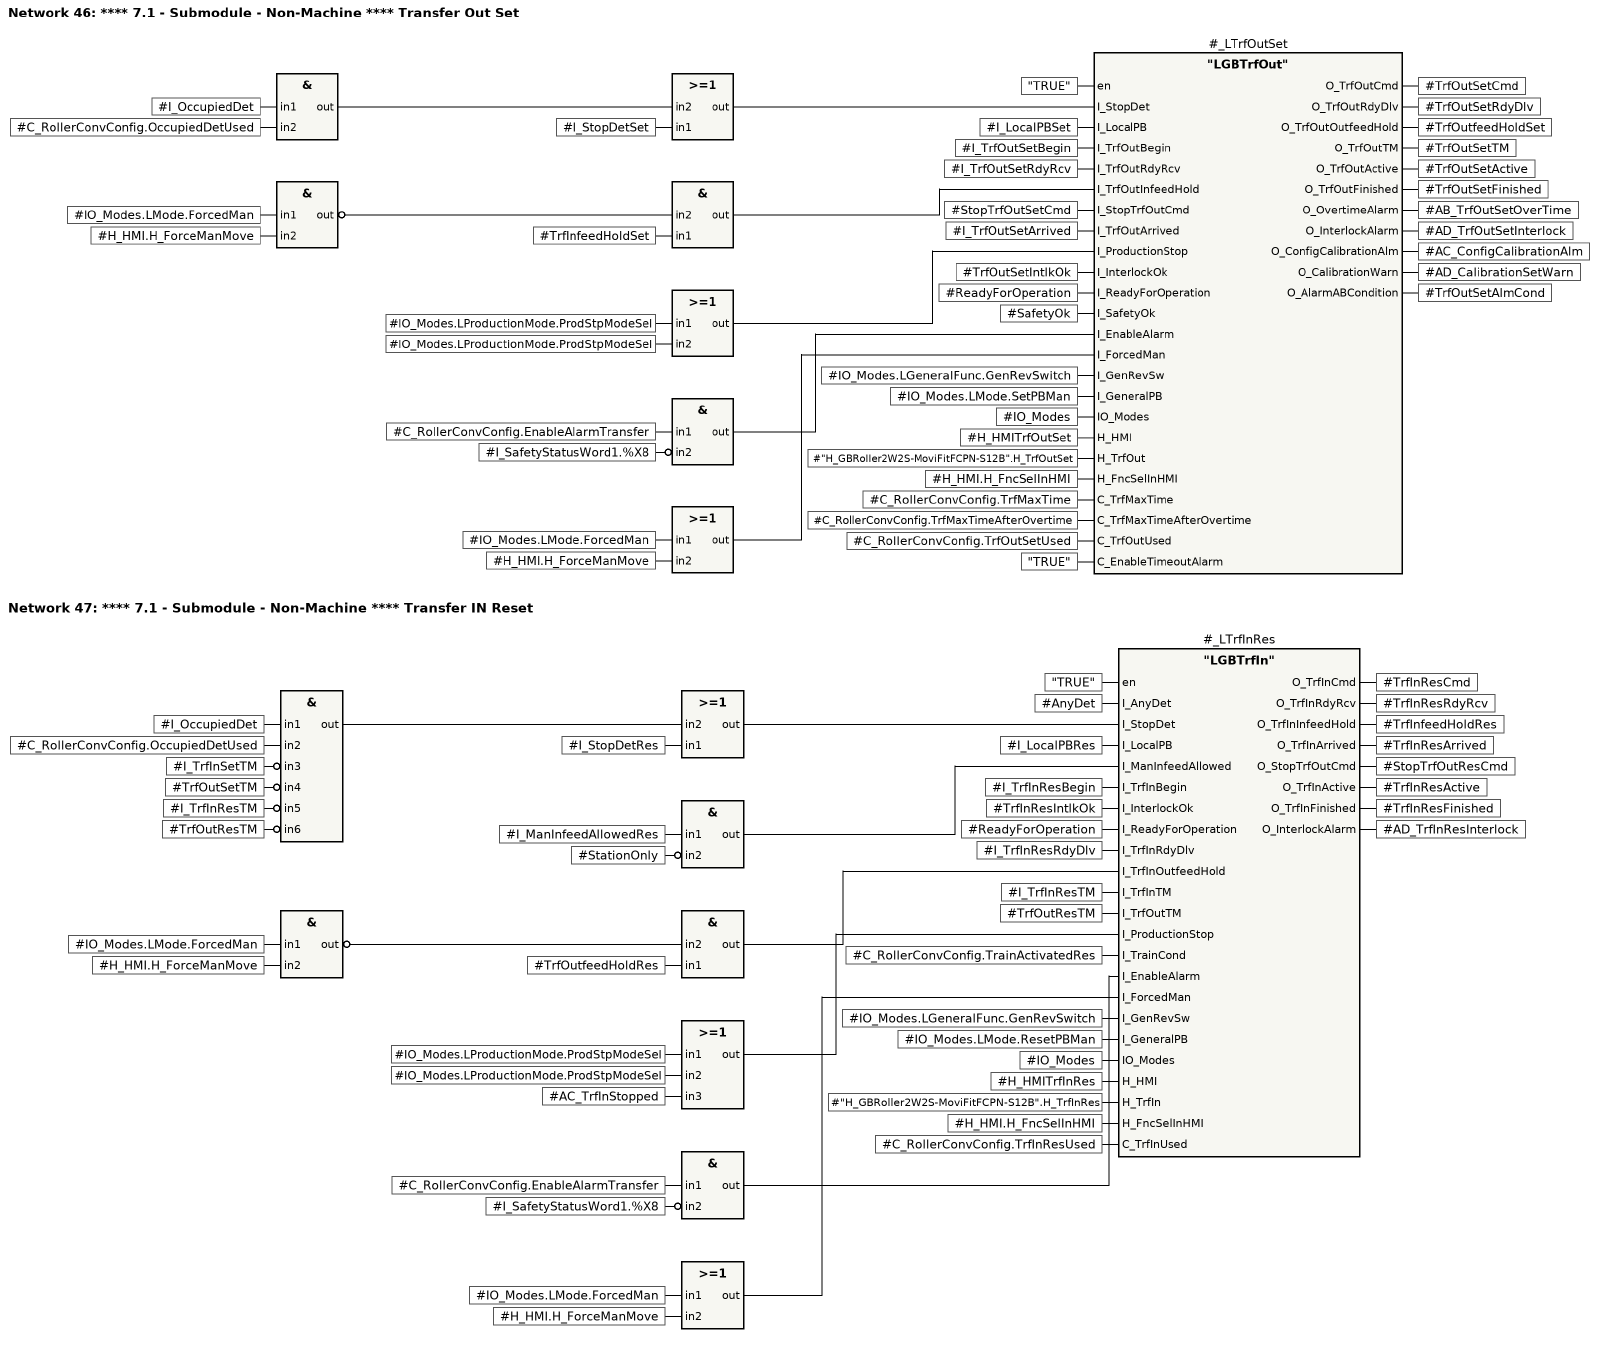
   IF "TRUE" THEN
       #_LTrfOutSet(I_StopDet := (#I_OccupiedDet AND #C_RollerConvConfig.OccupiedDetUsed) OR #I_StopDetSet,   // "LGBTrfOut"
                    I_LocalPB := #I_LocalPBSet,
                    I_TrfOutBegin := #I_TrfOutSetBegin,
                    I_TrfOutRdyRcv := #I_TrfOutSetRdyRcv,
                    I_TrfOutInfeedHold := NOT (#IO_Modes.LMode.ForcedMan AND #H_HMI.H_ForceManMove) AND #TrfInfeedHoldSet,
                    I_StopTrfOutCmd := #StopTrfOutSetCmd,
                    I_TrfOutArrived := #I_TrfOutSetArrived,
                    I_ProductionStop := #IO_Modes.LProductionMode.ProdStpModeSel OR #IO_Modes.LProductionMode.ProdStpModeSel,
                    I_InterlockOk := #TrfOutSetIntlkOk,
                    I_ReadyForOperation := #ReadyForOperation,
                    I_SafetyOk := #SafetyOk,
                    I_EnableAlarm := #C_RollerConvConfig.EnableAlarmTransfer AND NOT #I_SafetyStatusWord1.%X8,
                    I_ForcedMan := #IO_Modes.LMode.ForcedMan OR #H_HMI.H_ForceManMove,
                    I_GenRevSw := #IO_Modes.LGeneralFunc.GenRevSwitch,
                    I_GeneralPB := #IO_Modes.LMode.SetPBMan,
                    IO_Modes := #IO_Modes,
                    H_HMI := #H_HMITrfOutSet,
                    H_TrfOut := #"H_GBRoller2W2S-MoviFitFCPN-S12B".H_TrfOutSet,
                    H_FncSelInHMI := #H_HMI.H_FncSelInHMI,
                    C_TrfMaxTime := #C_RollerConvConfig.TrfMaxTime,
                    C_TrfMaxTimeAfterOvertime := #C_RollerConvConfig.TrfMaxTimeAfterOvertime,
                    C_TrfOutUsed := #C_RollerConvConfig.TrfOutSetUsed,
                    C_EnableTimeoutAlarm := "TRUE",
                    O_TrfOutCmd => #TrfOutSetCmd,
                    O_TrfOutRdyDlv => #TrfOutSetRdyDlv,
                    O_TrfOutOutfeedHold => #TrfOutfeedHoldSet,
                    O_TrfOutTM => #TrfOutSetTM,
                    O_TrfOutActive => #TrfOutSetActive,
                    O_TrfOutFinished => #TrfOutSetFinished,
                    O_OvertimeAlarm => #AB_TrfOutSetOverTime,
                    O_InterlockAlarm => #AD_TrfOutSetInterlock,
                    O_ConfigCalibrationAlm => #AC_ConfigCalibrationAlm,
                    O_CalibrationWarn => #AD_CalibrationSetWarn,
                    O_AlarmABCondition => #TrfOutSetAlmCond);
   END_IF;
END_REGION

REGION Network 47: **** 7.1 - Submodule - Non-Machine **** Transfer IN Reset
   // Transfer IN Reset
   IF "TRUE" THEN
       #_LTrfInRes(I_AnyDet := #AnyDet,   // "LGBTrfIn"
                   I_StopDet := (#I_OccupiedDet AND #C_RollerConvConfig.OccupiedDetUsed AND NOT #I_TrfInSetTM AND NOT #TrfOutSetTM AND NOT #I_TrfInResTM AND NOT #TrfOutResTM) OR #I_StopDetRes,
                   I_LocalPB := #I_LocalPBRes,
                   I_ManInfeedAllowed := #I_ManInfeedAllowedRes AND NOT #StationOnly,
                   I_TrfInBegin := #I_TrfInResBegin,
                   I_InterlockOk := #TrfInResIntlkOk,
                   I_ReadyForOperation := #ReadyForOperation,
                   I_TrfInRdyDlv := #I_TrfInResRdyDlv,
                   I_TrfInOutfeedHold := NOT (#IO_Modes.LMode.ForcedMan AND #H_HMI.H_ForceManMove) AND #TrfOutfeedHoldRes,
                   I_TrfInTM := #I_TrfInResTM,
                   I_TrfOutTM := #TrfOutResTM,
                   I_ProductionStop := #IO_Modes.LProductionMode.ProdStpModeSel OR #IO_Modes.LProductionMode.ProdStpModeSel OR #AC_TrfInStopped,
                   I_TrainCond := #C_RollerConvConfig.TrainActivatedRes,
                   I_EnableAlarm := #C_RollerConvConfig.EnableAlarmTransfer AND NOT #I_SafetyStatusWord1.%X8,
                   I_ForcedMan := #IO_Modes.LMode.ForcedMan OR #H_HMI.H_ForceManMove,
                   I_GenRevSw := #IO_Modes.LGeneralFunc.GenRevSwitch,
                   I_GeneralPB := #IO_Modes.LMode.ResetPBMan,
                   IO_Modes := #IO_Modes,
                   H_HMI := #H_HMITrfInRes,
                   H_TrfIn := #"H_GBRoller2W2S-MoviFitFCPN-S12B".H_TrfInRes,
                   H_FncSelInHMI := #H_HMI.H_FncSelInHMI,
                   C_TrfInUsed := #C_RollerConvConfig.TrfInResUsed,
                   O_TrfInCmd => #TrfInResCmd,
                   O_TrfInRdyRcv => #TrfInResRdyRcv,
                   O_TrfInInfeedHold => #TrfInfeedHoldRes,
                   O_TrfInArrived => #TrfInResArrived,
                   O_StopTrfOutCmd => #StopTrfOutResCmd,
                   O_TrfInActive => #TrfInResActive,
                   O_TrfInFinished => #TrfInResFinished,
                   O_InterlockAlarm => #AD_TrfInResInterlock);
   END_IF;
END_REGION

REGION Network 48: **** 7.1 - Submodule - Non-Machine **** Transfer Out Reset
   // Transfer Out Reset
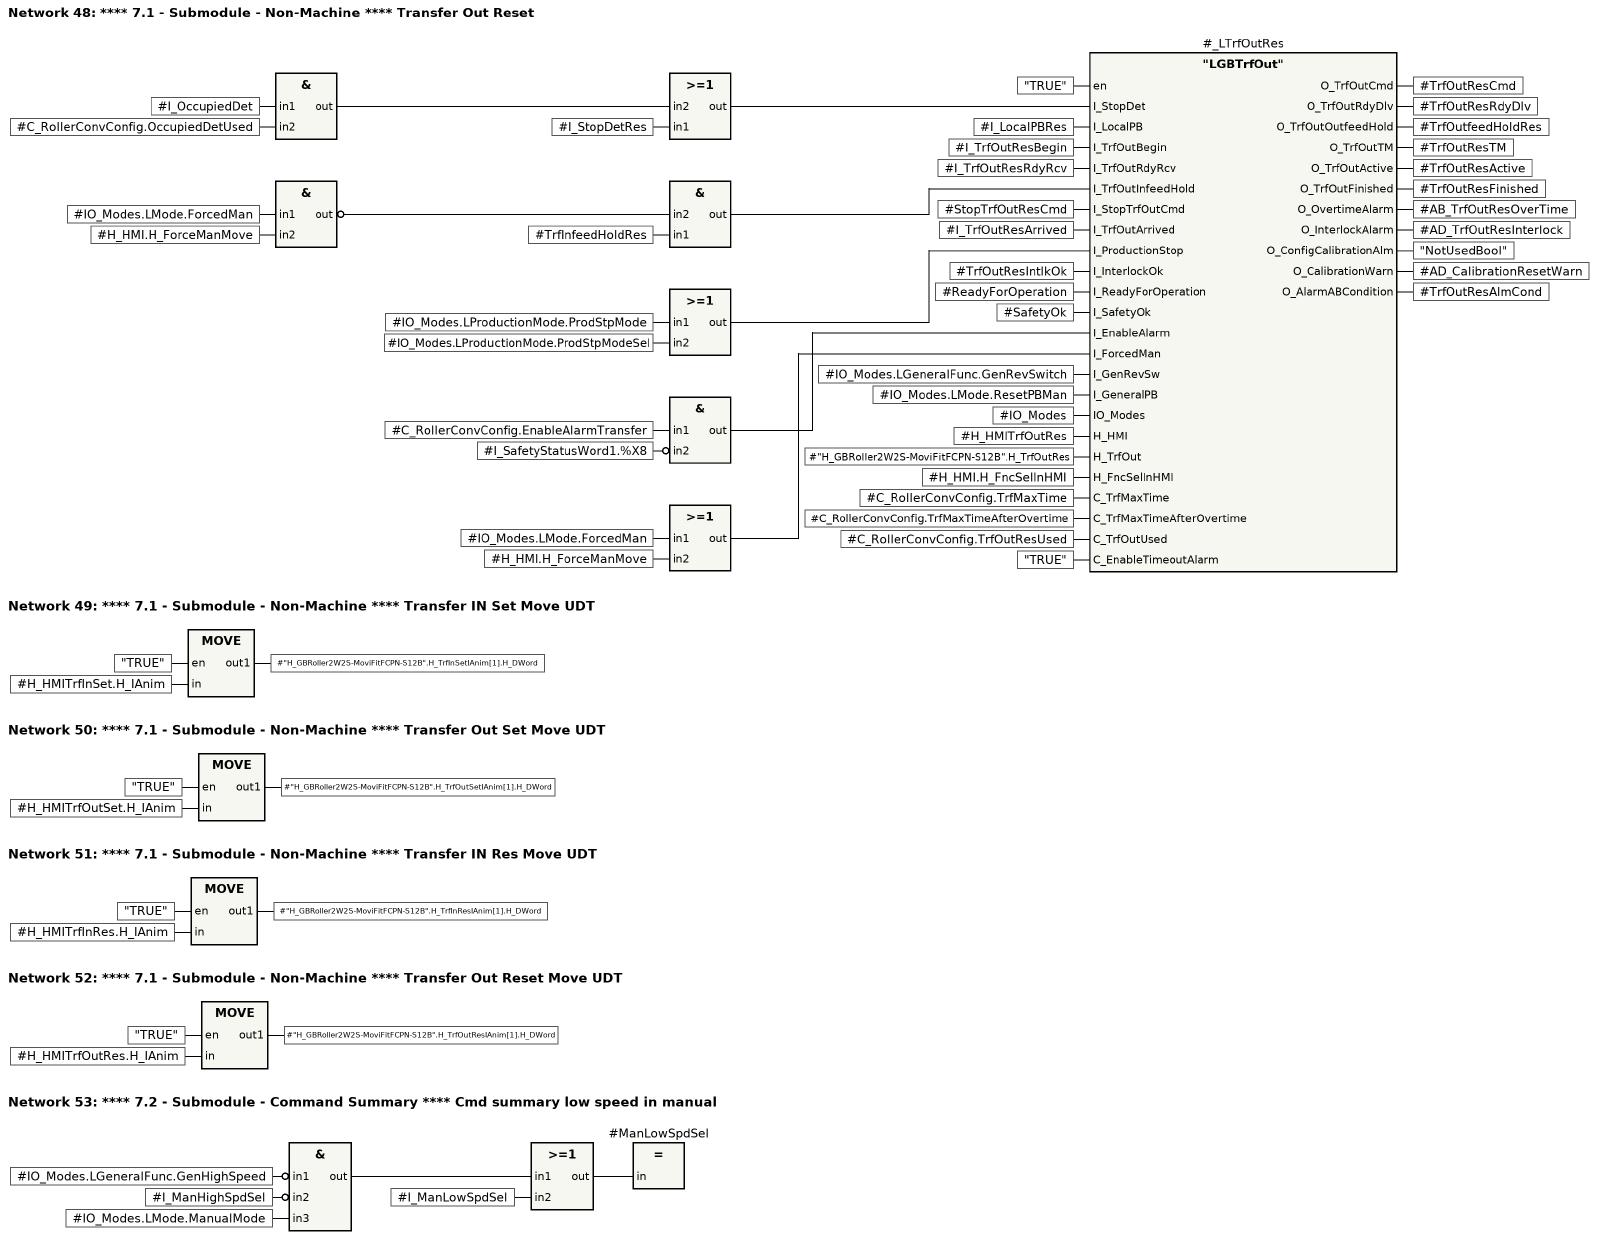
   IF "TRUE" THEN
       #_LTrfOutRes(I_StopDet := (#I_OccupiedDet AND #C_RollerConvConfig.OccupiedDetUsed) OR #I_StopDetRes,   // "LGBTrfOut"
                    I_LocalPB := #I_LocalPBRes,
                    I_TrfOutBegin := #I_TrfOutResBegin,
                    I_TrfOutRdyRcv := #I_TrfOutResRdyRcv,
                    I_TrfOutInfeedHold := NOT (#IO_Modes.LMode.ForcedMan AND #H_HMI.H_ForceManMove) AND #TrfInfeedHoldRes,
                    I_StopTrfOutCmd := #StopTrfOutResCmd,
                    I_TrfOutArrived := #I_TrfOutResArrived,
                    I_ProductionStop := #IO_Modes.LProductionMode.ProdStpMode OR #IO_Modes.LProductionMode.ProdStpModeSel,
                    I_InterlockOk := #TrfOutResIntlkOk,
                    I_ReadyForOperation := #ReadyForOperation,
                    I_SafetyOk := #SafetyOk,
                    I_EnableAlarm := #C_RollerConvConfig.EnableAlarmTransfer AND NOT #I_SafetyStatusWord1.%X8,
                    I_ForcedMan := #IO_Modes.LMode.ForcedMan OR #H_HMI.H_ForceManMove,
                    I_GenRevSw := #IO_Modes.LGeneralFunc.GenRevSwitch,
                    I_GeneralPB := #IO_Modes.LMode.ResetPBMan,
                    IO_Modes := #IO_Modes,
                    H_HMI := #H_HMITrfOutRes,
                    H_TrfOut := #"H_GBRoller2W2S-MoviFitFCPN-S12B".H_TrfOutRes,
                    H_FncSelInHMI := #H_HMI.H_FncSelInHMI,
                    C_TrfMaxTime := #C_RollerConvConfig.TrfMaxTime,
                    C_TrfMaxTimeAfterOvertime := #C_RollerConvConfig.TrfMaxTimeAfterOvertime,
                    C_TrfOutUsed := #C_RollerConvConfig.TrfOutResUsed,
                    C_EnableTimeoutAlarm := "TRUE",
                    O_TrfOutCmd => #TrfOutResCmd,
                    O_TrfOutRdyDlv => #TrfOutResRdyDlv,
                    O_TrfOutOutfeedHold => #TrfOutfeedHoldRes,
                    O_TrfOutTM => #TrfOutResTM,
                    O_TrfOutActive => #TrfOutResActive,
                    O_TrfOutFinished => #TrfOutResFinished,
                    O_OvertimeAlarm => #AB_TrfOutResOverTime,
                    O_InterlockAlarm => #AD_TrfOutResInterlock,
                    O_ConfigCalibrationAlm => "NotUsedBool",
                    O_CalibrationWarn => #AD_CalibrationResetWarn,
                    O_AlarmABCondition => #TrfOutResAlmCond);
   END_IF;
END_REGION

REGION Network 49: **** 7.1 - Submodule - Non-Machine **** Transfer IN Set Move UDT
   // Transfer IN Set Move UDT
   IF "TRUE" THEN
       #"H_GBRoller2W2S-MoviFitFCPN-S12B".H_TrfInSetIAnim[1].H_DWord := #H_HMITrfInSet.H_IAnim;
   END_IF;
END_REGION

REGION Network 50: **** 7.1 - Submodule - Non-Machine **** Transfer Out Set Move UDT
   // Transfer Out Set Move UDT
   IF "TRUE" THEN
       #"H_GBRoller2W2S-MoviFitFCPN-S12B".H_TrfOutSetIAnim[1].H_DWord := #H_HMITrfOutSet.H_IAnim;
   END_IF;
END_REGION

REGION Network 51: **** 7.1 - Submodule - Non-Machine **** Transfer IN Res Move UDT
   // Transfer IN Res Move UDT
   IF "TRUE" THEN
       #"H_GBRoller2W2S-MoviFitFCPN-S12B".H_TrfInResIAnim[1].H_DWord := #H_HMITrfInRes.H_IAnim;
   END_IF;
END_REGION

REGION Network 52: **** 7.1 - Submodule - Non-Machine **** Transfer Out Reset Move UDT
   // Transfer Out Reset Move UDT
   IF "TRUE" THEN
       #"H_GBRoller2W2S-MoviFitFCPN-S12B".H_TrfOutResIAnim[1].H_DWord := #H_HMITrfOutRes.H_IAnim;
   END_IF;
END_REGION

REGION Network 53: **** 7.2 - Submodule - Command Summary **** Cmd summary low speed in manual
   // Cmd summary low speed in manual
   #ManLowSpdSel := (NOT #IO_Modes.LGeneralFunc.GenHighSpeed AND NOT #I_ManHighSpdSel AND #IO_Modes.LMode.ManualMode) OR #I_ManLowSpdSel;
END_REGION

REGION Network 54: **** 7.2 - Submodule - Command Summary **** Motor Command Low Speed Set
   // Motor Command Low Speed Set
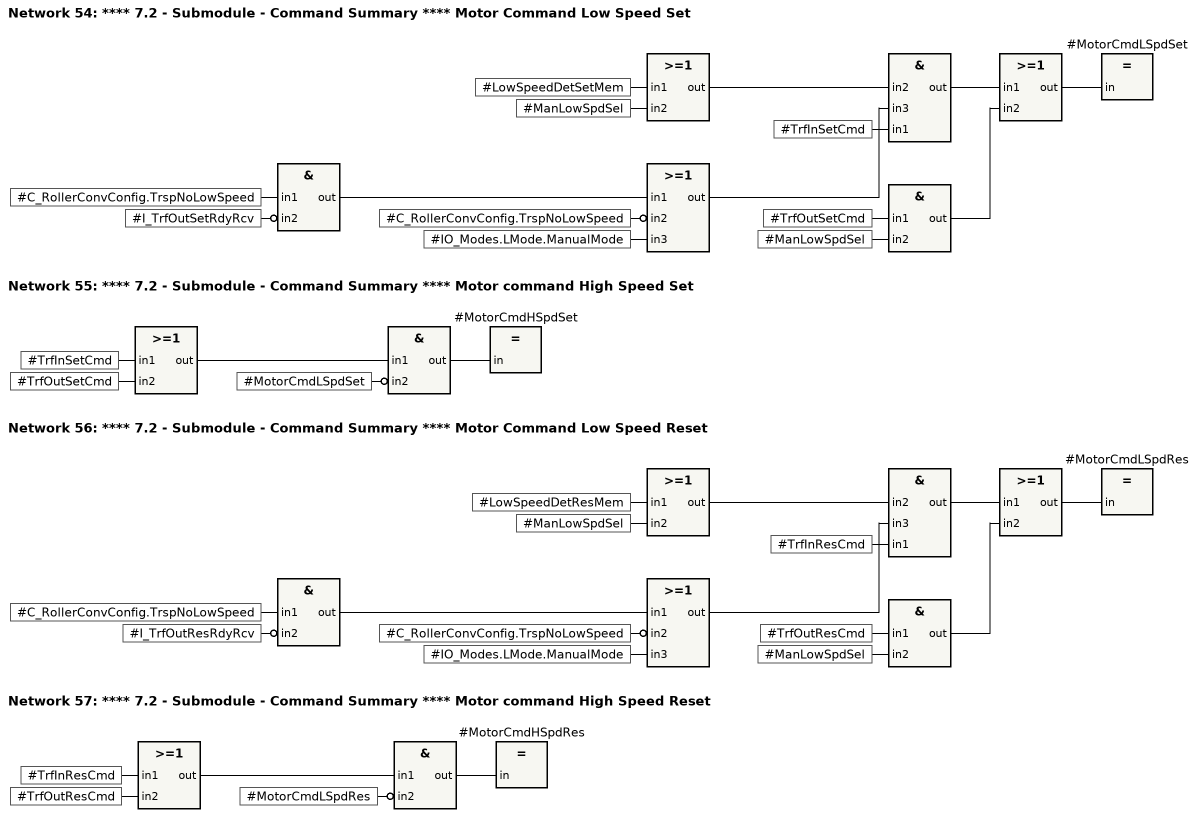
   #MotorCmdLSpdSet := ((#LowSpeedDetSetMem OR #ManLowSpdSel) AND ((#C_RollerConvConfig.TrspNoLowSpeed AND NOT #I_TrfOutSetRdyRcv) OR NOT #C_RollerConvConfig.TrspNoLowSpeed OR #IO_Modes.LMode.ManualMode) AND #TrfInSetCmd) OR (#TrfOutSetCmd AND #ManLowSpdSel);
END_REGION

REGION Network 55: **** 7.2 - Submodule - Command Summary **** Motor command High Speed Set
   // Motor command High Speed Set
   #MotorCmdHSpdSet := (#TrfInSetCmd OR #TrfOutSetCmd) AND NOT #MotorCmdLSpdSet;
END_REGION

REGION Network 56: **** 7.2 - Submodule - Command Summary **** Motor Command Low Speed Reset
   // Motor Command Low Speed Reset
   #MotorCmdLSpdRes := ((#LowSpeedDetResMem OR #ManLowSpdSel) AND ((#C_RollerConvConfig.TrspNoLowSpeed AND NOT #I_TrfOutResRdyRcv) OR NOT #C_RollerConvConfig.TrspNoLowSpeed OR #IO_Modes.LMode.ManualMode) AND #TrfInResCmd) OR (#TrfOutResCmd AND #ManLowSpdSel);
END_REGION

REGION Network 57: **** 7.2 - Submodule - Command Summary **** Motor command High Speed Reset
   // Motor command High Speed Reset
   #MotorCmdHSpdRes := (#TrfInResCmd OR #TrfOutResCmd) AND NOT #MotorCmdLSpdRes;
END_REGION

REGION Network 58: **** 7.3 - Submodule - Machine **** Motor loop MOVIFIT-FC
   // Motor loop MOVIFIT-FC
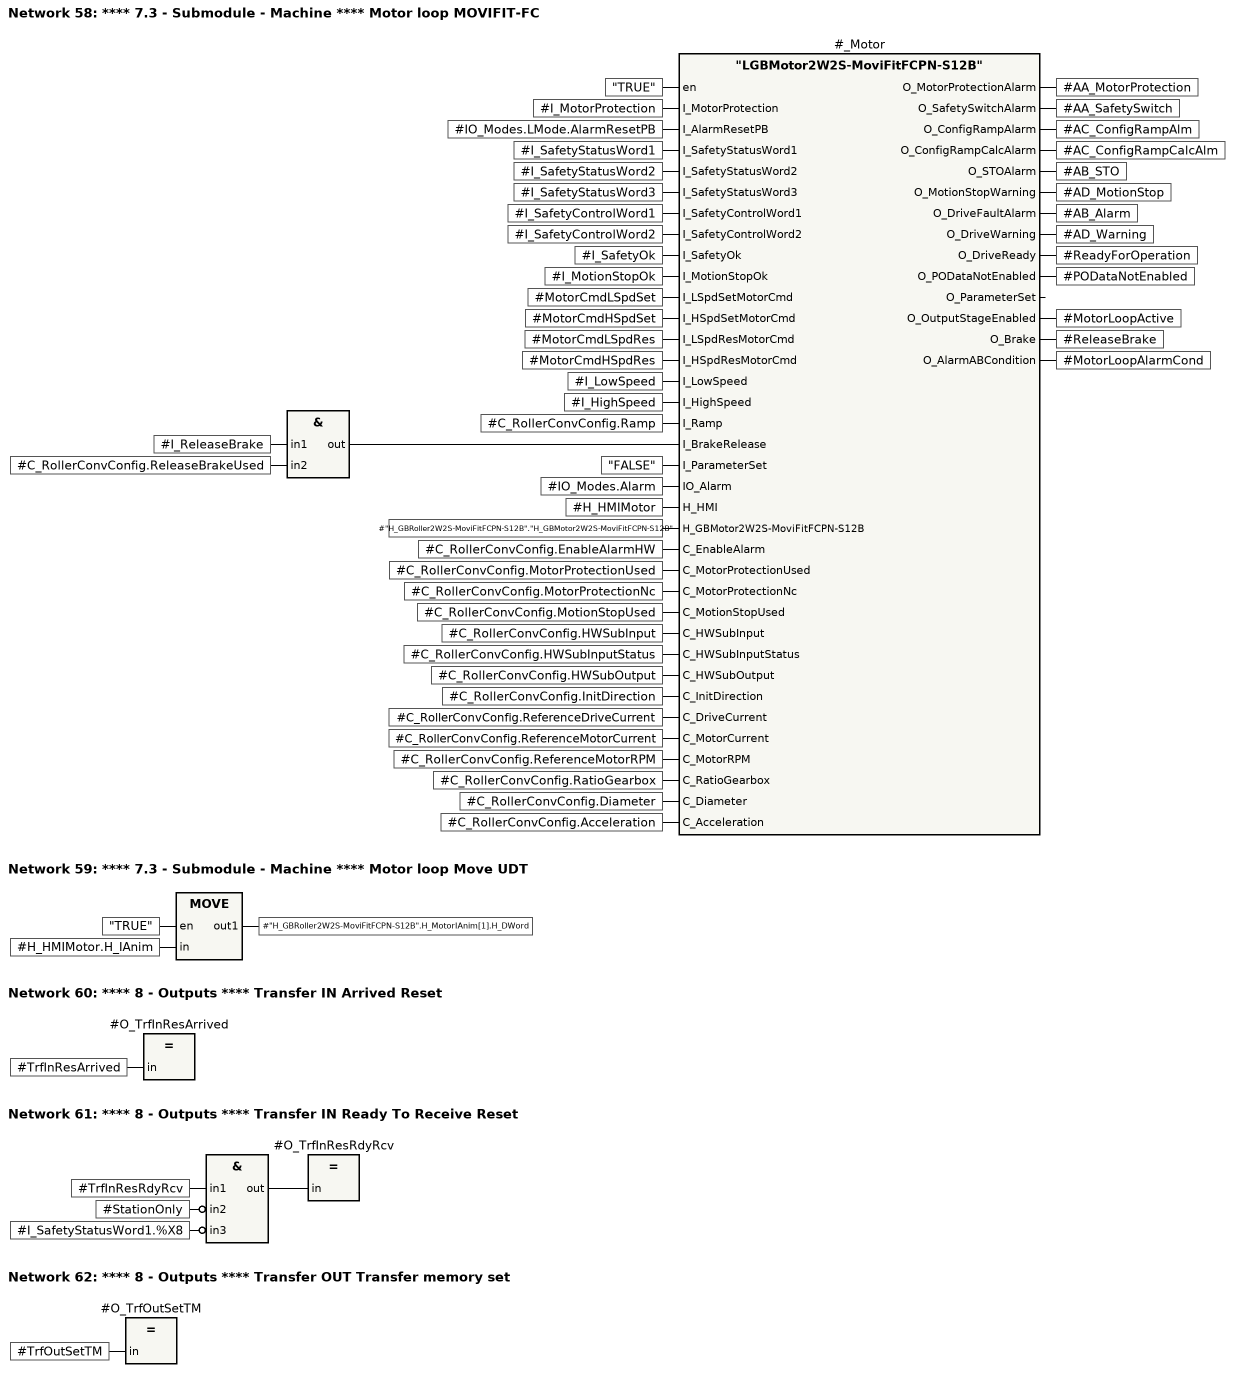
   IF "TRUE" THEN
       #_Motor(I_MotorProtection := #I_MotorProtection,   // "LGBMotor2W2S-MoviFitFCPN-S12B"
               I_AlarmResetPB := #IO_Modes.LMode.AlarmResetPB,
               I_SafetyStatusWord1 := #I_SafetyStatusWord1,
               I_SafetyStatusWord2 := #I_SafetyStatusWord2,
               I_SafetyStatusWord3 := #I_SafetyStatusWord3,
               I_SafetyControlWord1 := #I_SafetyControlWord1,
               I_SafetyControlWord2 := #I_SafetyControlWord2,
               I_SafetyOk := #I_SafetyOk,
               I_MotionStopOk := #I_MotionStopOk,
               I_LSpdSetMotorCmd := #MotorCmdLSpdSet,
               I_HSpdSetMotorCmd := #MotorCmdHSpdSet,
               I_LSpdResMotorCmd := #MotorCmdLSpdRes,
               I_HSpdResMotorCmd := #MotorCmdHSpdRes,
               I_LowSpeed := #I_LowSpeed,
               I_HighSpeed := #I_HighSpeed,
               I_Ramp := #C_RollerConvConfig.Ramp,
               I_BrakeRelease := #I_ReleaseBrake AND #C_RollerConvConfig.ReleaseBrakeUsed,
               I_ParameterSet := "FALSE",
               IO_Alarm := #IO_Modes.Alarm,
               H_HMI := #H_HMIMotor,
               "H_GBMotor2W2S-MoviFitFCPN-S12B" := #"H_GBRoller2W2S-MoviFitFCPN-S12B"."H_GBMotor2W2S-MoviFitFCPN-S12B",
               C_EnableAlarm := #C_RollerConvConfig.EnableAlarmHW,
               C_MotorProtectionUsed := #C_RollerConvConfig.MotorProtectionUsed,
               C_MotorProtectionNc := #C_RollerConvConfig.MotorProtectionNc,
               C_MotionStopUsed := #C_RollerConvConfig.MotionStopUsed,
               C_HWSubInput := #C_RollerConvConfig.HWSubInput,
               C_HWSubInputStatus := #C_RollerConvConfig.HWSubInputStatus,
               C_HWSubOutput := #C_RollerConvConfig.HWSubOutput,
               C_InitDirection := #C_RollerConvConfig.InitDirection,
               C_DriveCurrent := #C_RollerConvConfig.ReferenceDriveCurrent,
               C_MotorCurrent := #C_RollerConvConfig.ReferenceMotorCurrent,
               C_MotorRPM := #C_RollerConvConfig.ReferenceMotorRPM,
               C_RatioGearbox := #C_RollerConvConfig.RatioGearbox,
               C_Diameter := #C_RollerConvConfig.Diameter,
               C_Acceleration := #C_RollerConvConfig.Acceleration,
               O_MotorProtectionAlarm => #AA_MotorProtection,
               O_SafetySwitchAlarm => #AA_SafetySwitch,
               O_ConfigRampAlarm => #AC_ConfigRampAlm,
               O_ConfigRampCalcAlarm => #AC_ConfigRampCalcAlm,
               O_STOAlarm => #AB_STO,
               O_MotionStopWarning => #AD_MotionStop,
               O_DriveFaultAlarm => #AB_Alarm,
               O_DriveWarning => #AD_Warning,
               O_DriveReady => #ReadyForOperation,
               O_PODataNotEnabled => #PODataNotEnabled,
               O_OutputStageEnabled => #MotorLoopActive,
               O_Brake => #ReleaseBrake,
               O_AlarmABCondition => #MotorLoopAlarmCond);
   END_IF;
END_REGION

REGION Network 59: **** 7.3 - Submodule - Machine **** Motor loop Move UDT
   IF "TRUE" THEN #"H_GBRoller2W2S-MoviFitFCPN-S12B".H_MotorIAnim[1].H_DWord := #H_HMIMotor.H_IAnim; END_IF;
END_REGION

REGION Network 60: **** 8 - Outputs **** Transfer IN Arrived Reset
   // Transfer IN Arrived Reset
   #O_TrfInResArrived := #TrfInResArrived;
END_REGION

REGION Network 61: **** 8 - Outputs **** Transfer IN Ready To Receive Reset
   // Transfer IN Ready To Receive Reset
   #O_TrfInResRdyRcv := #TrfInResRdyRcv AND NOT #StationOnly AND NOT #I_SafetyStatusWord1.%X8;
END_REGION

REGION Network 62: **** 8 - Outputs **** Transfer OUT Transfer memory set
   // Transfer OUT Transfer memory set
   #O_TrfOutSetTM := #TrfOutSetTM;
END_REGION

REGION Network 63: **** 8 - Outputs **** Transfer OUT Ready To Deliver set
   // Transfer OUT Ready To Deliver set
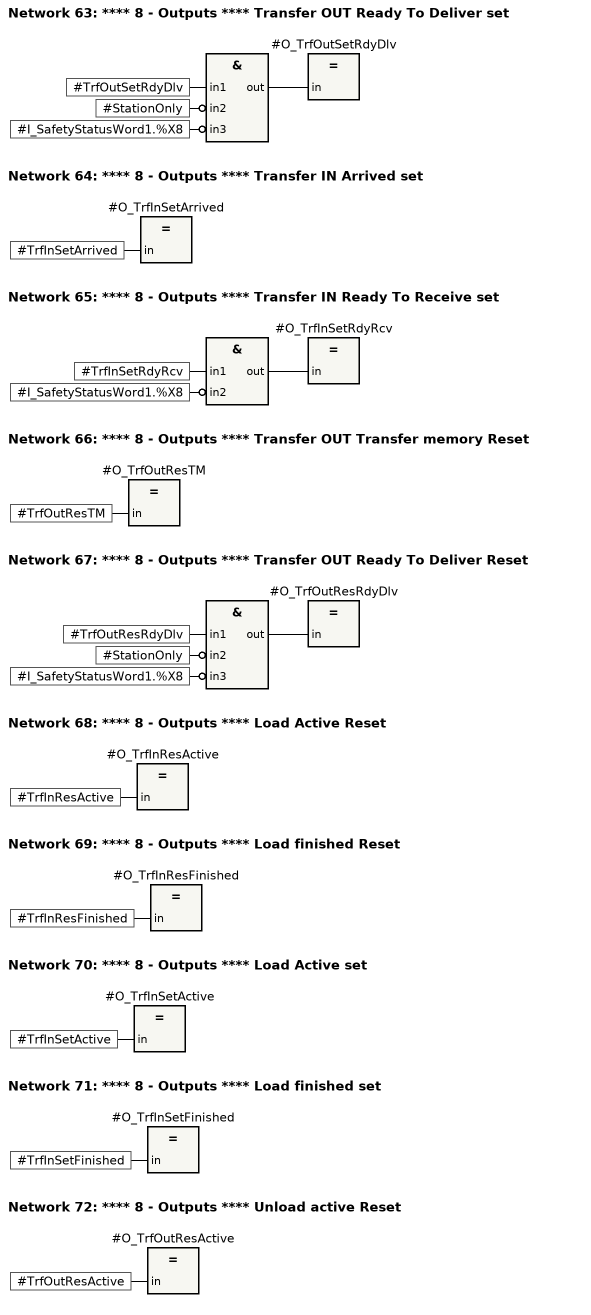
   #O_TrfOutSetRdyDlv := #TrfOutSetRdyDlv AND NOT #StationOnly AND NOT #I_SafetyStatusWord1.%X8;
END_REGION

REGION Network 64: **** 8 - Outputs **** Transfer IN Arrived set
   // Transfer IN Arrived set
   #O_TrfInSetArrived := #TrfInSetArrived;
END_REGION

REGION Network 65: **** 8 - Outputs **** Transfer IN Ready To Receive set
   // Transfer IN Ready To Receive set
   #O_TrfInSetRdyRcv := #TrfInSetRdyRcv AND NOT #I_SafetyStatusWord1.%X8;
END_REGION

REGION Network 66: **** 8 - Outputs **** Transfer OUT Transfer memory Reset
   // Transfer OUT Transfer memory Reset
   #O_TrfOutResTM := #TrfOutResTM;
END_REGION

REGION Network 67: **** 8 - Outputs **** Transfer OUT Ready To Deliver Reset
   // Transfer OUT Ready To Deliver Reset
   #O_TrfOutResRdyDlv := #TrfOutResRdyDlv AND NOT #StationOnly AND NOT #I_SafetyStatusWord1.%X8;
END_REGION

REGION Network 68: **** 8 - Outputs **** Load Active Reset
   // Load Active Reset
   #O_TrfInResActive := #TrfInResActive;
END_REGION

REGION Network 69: **** 8 - Outputs **** Load finished Reset
   // Load finished Reset
   #O_TrfInResFinished := #TrfInResFinished;
END_REGION

REGION Network 70: **** 8 - Outputs **** Load Active set
   // Load Active set
   #O_TrfInSetActive := #TrfInSetActive;
END_REGION

REGION Network 71: **** 8 - Outputs **** Load finished set
   // Load finished set
   #O_TrfInSetFinished := #TrfInSetFinished;
END_REGION

REGION Network 72: **** 8 - Outputs **** Unload active Reset
   // Unload active Reset
   #O_TrfOutResActive := #TrfOutResActive;
END_REGION

REGION Network 73: **** 8 - Outputs **** Unload finished Reset
   // Unload finished Reset
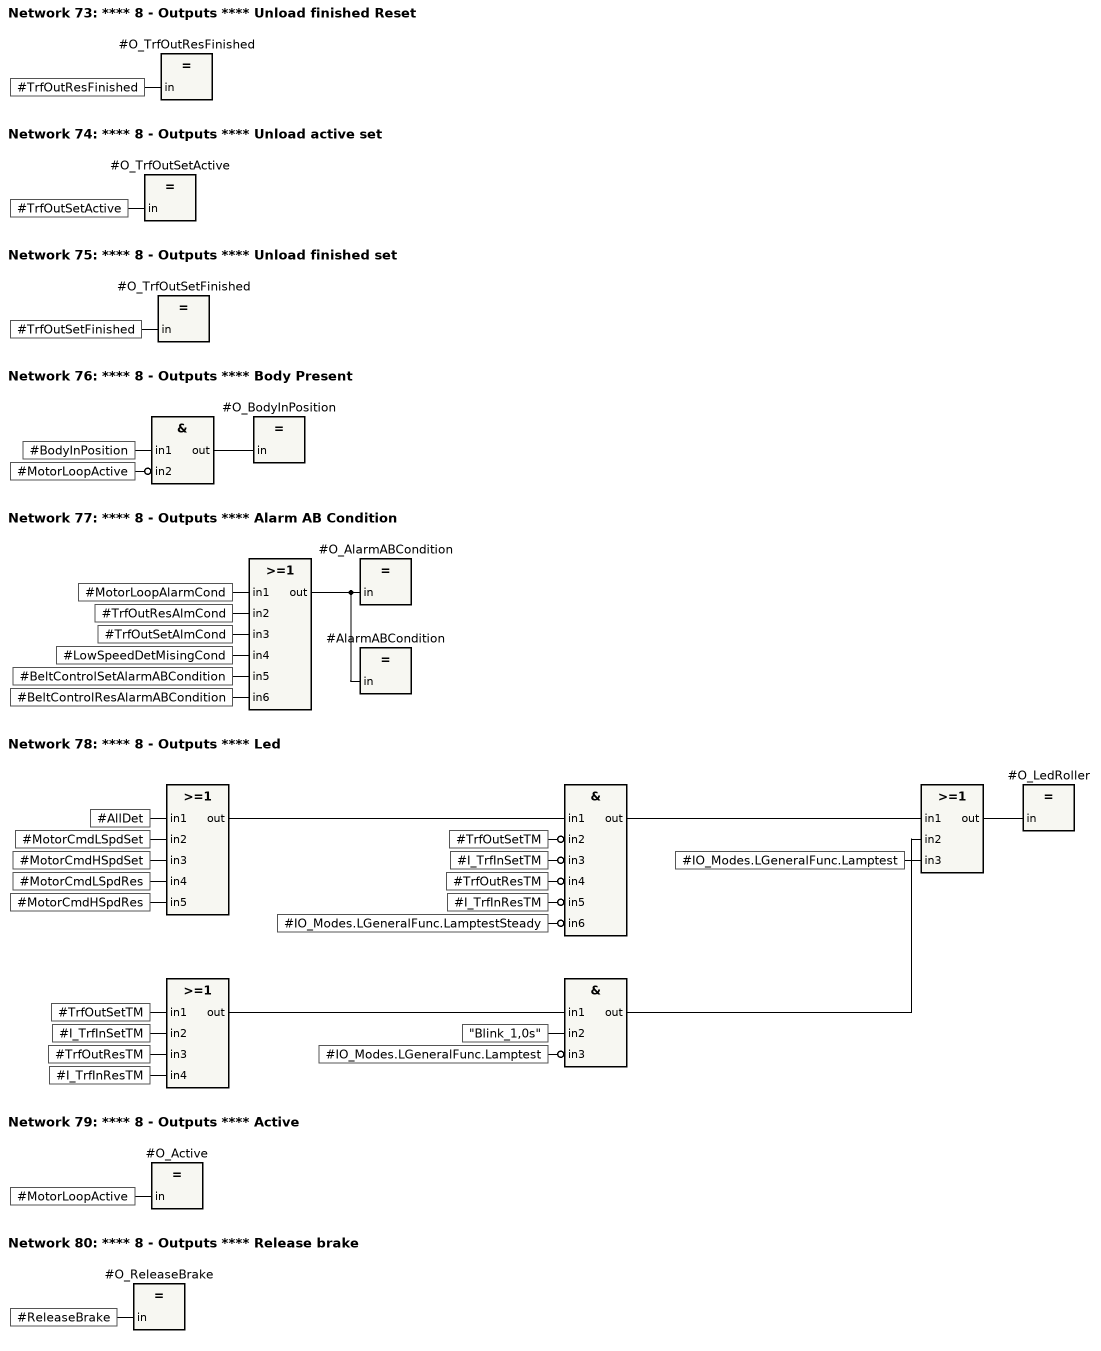
   #O_TrfOutResFinished := #TrfOutResFinished;
END_REGION

REGION Network 74: **** 8 - Outputs **** Unload active set
   // Unload active set
   #O_TrfOutSetActive := #TrfOutSetActive;
END_REGION

REGION Network 75: **** 8 - Outputs **** Unload finished set
   // Unload finished set
   #O_TrfOutSetFinished := #TrfOutSetFinished;
END_REGION

REGION Network 76: **** 8 - Outputs **** Body Present
   // Body present
   #O_BodyInPosition := #BodyInPosition AND NOT #MotorLoopActive;
END_REGION

REGION Network 77: **** 8 - Outputs **** Alarm AB Condition
   // Alarm AB Condition
   #O_AlarmABCondition := #MotorLoopAlarmCond OR #TrfOutResAlmCond OR #TrfOutSetAlmCond OR #LowSpeedDetMisingCond OR #BeltControlSetAlarmABCondition OR #BeltControlResAlarmABCondition;
   #AlarmABCondition := #O_AlarmABCondition;
END_REGION

REGION Network 78: **** 8 - Outputs **** Led
   // Led
   #O_LedRoller := ((#AllDet OR #MotorCmdLSpdSet OR #MotorCmdHSpdSet OR #MotorCmdLSpdRes OR #MotorCmdHSpdRes) AND NOT #TrfOutSetTM AND NOT #I_TrfInSetTM AND NOT #TrfOutResTM AND NOT #I_TrfInResTM AND NOT #IO_Modes.LGeneralFunc.LamptestSteady) OR ((#TrfOutSetTM OR #I_TrfInSetTM OR #TrfOutResTM OR #I_TrfInResTM) AND "Blink_1,0s" AND NOT #IO_Modes.LGeneralFunc.Lamptest) OR #IO_Modes.LGeneralFunc.Lamptest;
END_REGION

REGION Network 79: **** 8 - Outputs **** Active
   // Active
   #O_Active := #MotorLoopActive;
END_REGION

REGION Network 80: **** 8 - Outputs **** Release brake
   // Release brake
   #O_ReleaseBrake := #ReleaseBrake;
END_REGION

REGION Network 81: **** 8 - Outputs **** Occupied
   // Occupied
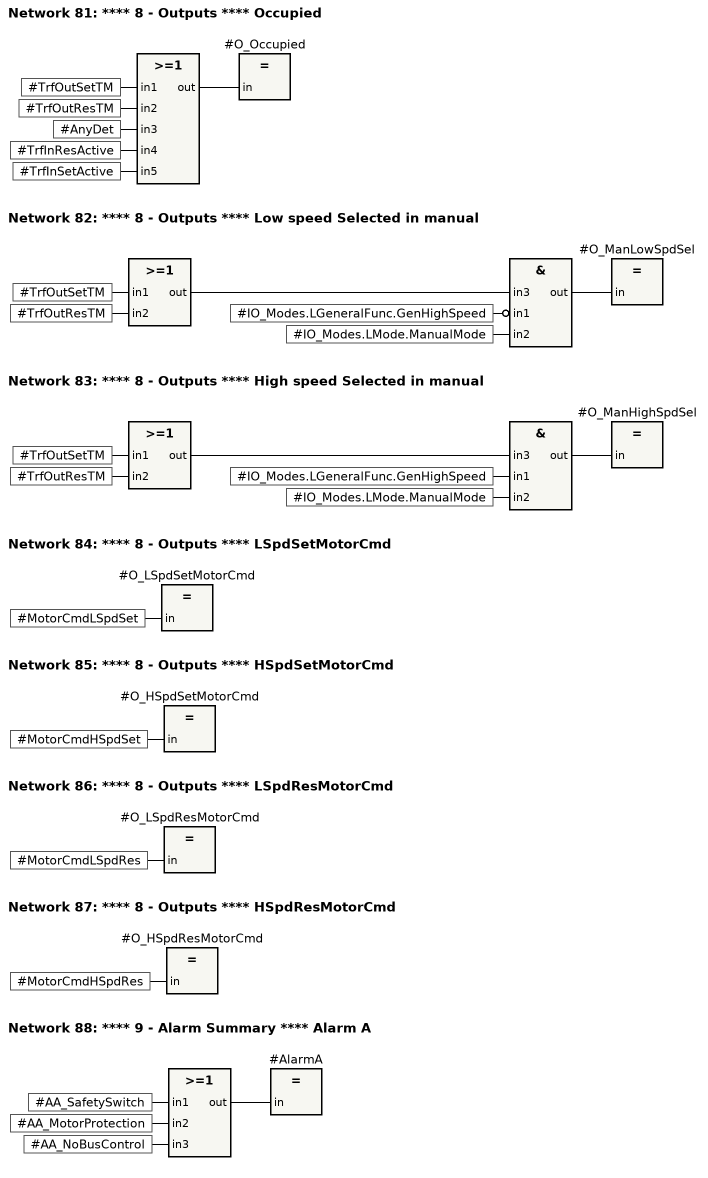
   #O_Occupied := #TrfOutSetTM OR #TrfOutResTM OR #AnyDet OR #TrfInResActive OR #TrfInSetActive;
END_REGION

REGION Network 82: **** 8 - Outputs **** Low speed Selected in manual
   #O_ManLowSpdSel := (#TrfOutSetTM OR #TrfOutResTM) AND NOT #IO_Modes.LGeneralFunc.GenHighSpeed AND #IO_Modes.LMode.ManualMode;
END_REGION

REGION Network 83: **** 8 - Outputs **** High speed Selected in manual
   #O_ManHighSpdSel := (#TrfOutSetTM OR #TrfOutResTM) AND #IO_Modes.LGeneralFunc.GenHighSpeed AND #IO_Modes.LMode.ManualMode;
END_REGION

REGION Network 84: **** 8 - Outputs **** LSpdSetMotorCmd
   // LSpdSetMotorCmd
   #O_LSpdSetMotorCmd := #MotorCmdLSpdSet;
END_REGION

REGION Network 85: **** 8 - Outputs **** HSpdSetMotorCmd
   // HSpdSetMotorCmd
   #O_HSpdSetMotorCmd := #MotorCmdHSpdSet;
END_REGION

REGION Network 86: **** 8 - Outputs **** LSpdResMotorCmd
   // LSpdResMotorCmd
   #O_LSpdResMotorCmd := #MotorCmdLSpdRes;
END_REGION

REGION Network 87: **** 8 - Outputs **** HSpdResMotorCmd
   // HSpdresMotorCmd
   #O_HSpdResMotorCmd := #MotorCmdHSpdRes;
END_REGION

REGION Network 88: **** 9 - Alarm Summary **** Alarm A
   // Alarm A
   #AlarmA := #AA_SafetySwitch OR #AA_MotorProtection OR #AA_NoBusControl;
END_REGION

REGION Network 89: **** 9 - Alarm Summary **** Alarm B
   // Alarm B
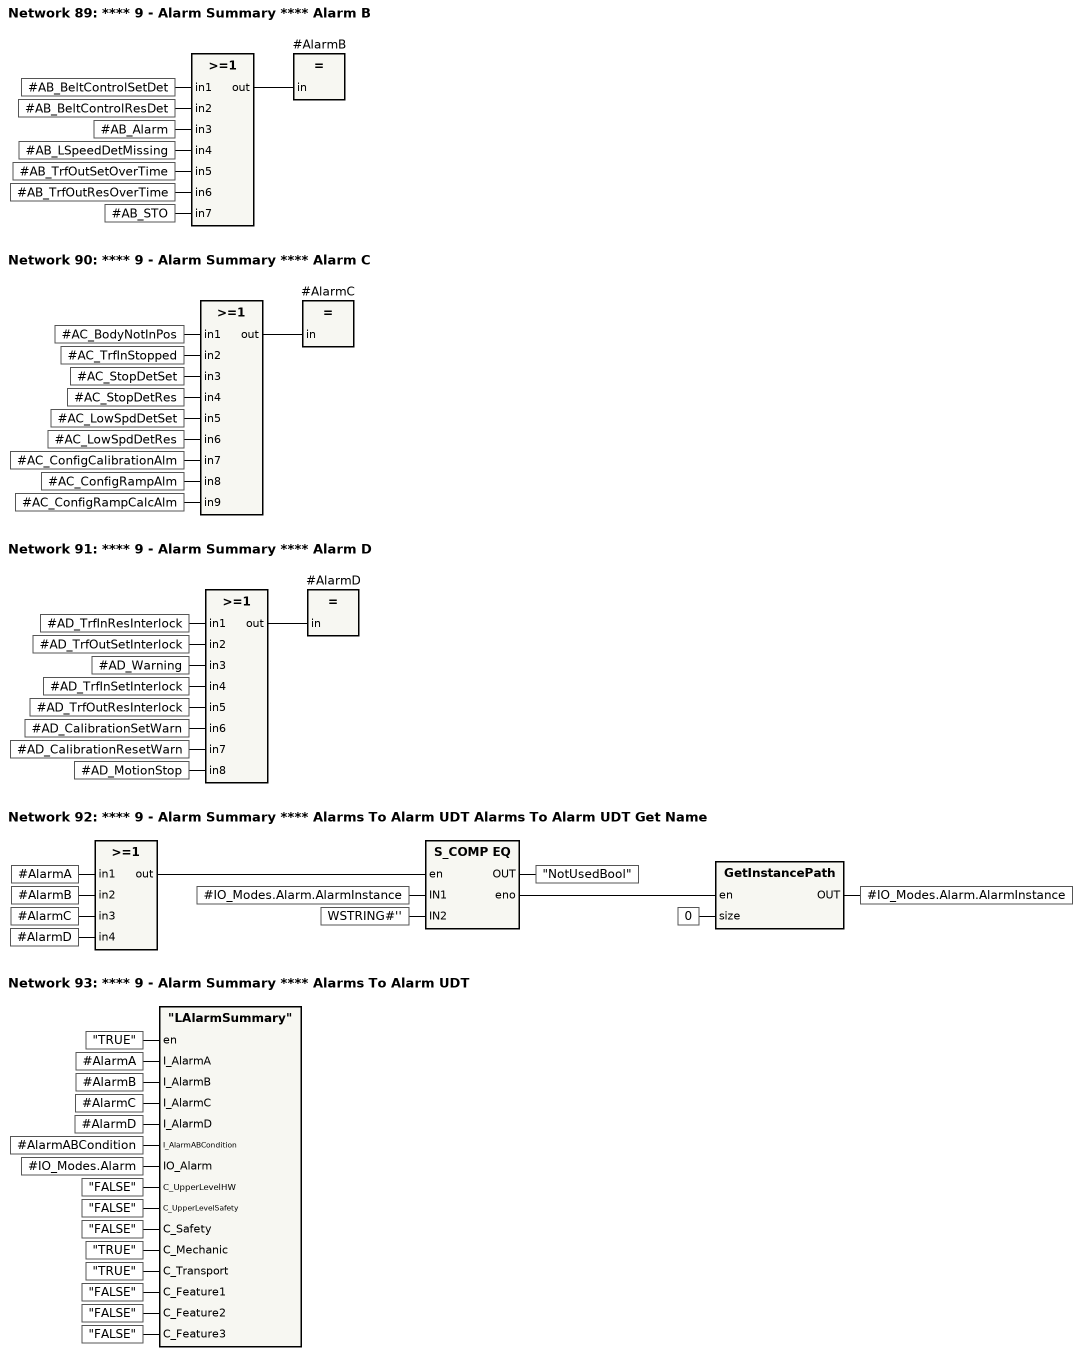
   #AlarmB := #AB_BeltControlSetDet OR #AB_BeltControlResDet OR #AB_Alarm OR #AB_LSpeedDetMissing OR #AB_TrfOutSetOverTime OR #AB_TrfOutResOverTime OR #AB_STO;
END_REGION

REGION Network 90: **** 9 - Alarm Summary **** Alarm C
   // Alarm C
   #AlarmC := #AC_BodyNotInPos OR #AC_TrfInStopped OR #AC_StopDetSet OR #AC_StopDetRes OR #AC_LowSpdDetSet OR #AC_LowSpdDetRes OR #AC_ConfigCalibrationAlm OR #AC_ConfigRampAlm OR #AC_ConfigRampCalcAlm;
END_REGION

REGION Network 91: **** 9 - Alarm Summary **** Alarm D
   // Alarm D
   #AlarmD := #AD_TrfInResInterlock OR #AD_TrfOutSetInterlock OR #AD_Warning OR #AD_TrfInSetInterlock OR #AD_TrfOutResInterlock OR #AD_CalibrationSetWarn OR #AD_CalibrationResetWarn OR #AD_MotionStop;
END_REGION

REGION Network 92: **** 9 - Alarm Summary **** Alarms To Alarm UDT Alarms To Alarm UDT Get Name
   // Alarm D
   S_COMP(EN := #AlarmA OR #AlarmB OR #AlarmC OR #AlarmD,
          IN1 := #IO_Modes.Alarm.AlarmInstance,
          IN2 := WSTRING#'',
          OUT => "NotUsedBool",
          ENO => #_w1);
   IF #_w1 THEN GetInstancePath(size := 0, OUT => #IO_Modes.Alarm.AlarmInstance); END_IF;
END_REGION

REGION Network 93: **** 9 - Alarm Summary **** Alarms To Alarm UDT
   // Alarm D
   IF "TRUE" THEN
       "LAlarmSummary"(I_AlarmA := #AlarmA,
                       I_AlarmB := #AlarmB,
                       I_AlarmC := #AlarmC,
                       I_AlarmD := #AlarmD,
                       I_AlarmABCondition := #AlarmABCondition,
                       IO_Alarm := #IO_Modes.Alarm,
                       C_UpperLevelHW := "FALSE",
                       C_UpperLevelSafety := "FALSE",
                       C_Safety := "FALSE",
                       C_Mechanic := "TRUE",
                       C_Transport := "TRUE",
                       C_Feature1 := "FALSE",
                       C_Feature2 := "FALSE",
                       C_Feature3 := "FALSE");
   END_IF;
END_REGION

REGION Network 94: **** 9.1 - Alarm Output **** Alarm A
   // Alarm A
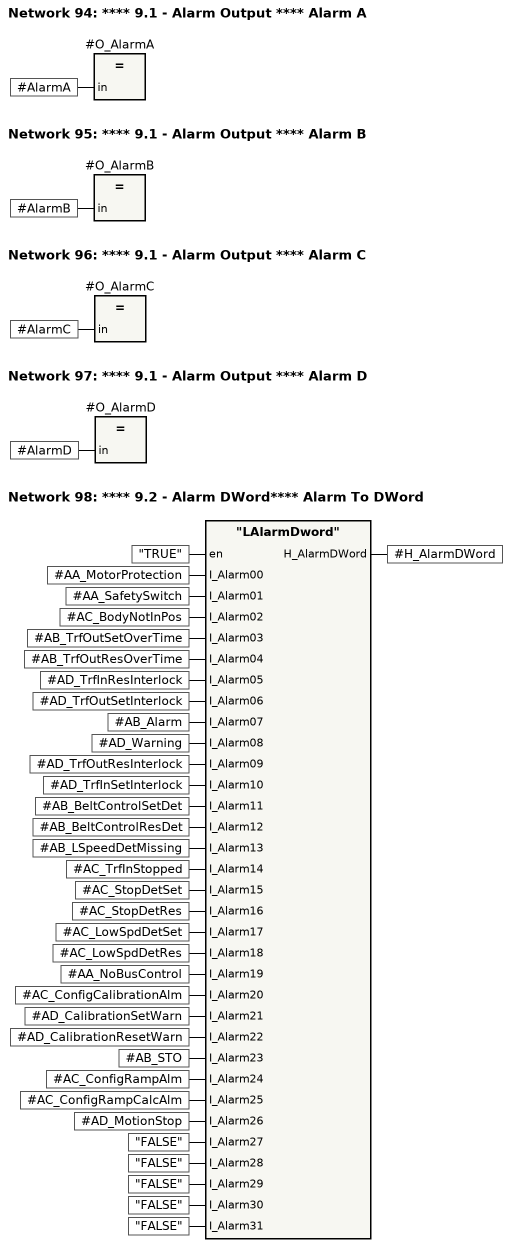
   #O_AlarmA := #AlarmA;
END_REGION

REGION Network 95: **** 9.1 - Alarm Output **** Alarm B
   // Alarm B
   #O_AlarmB := #AlarmB;
END_REGION

REGION Network 96: **** 9.1 - Alarm Output **** Alarm C
   // Alarm C
   #O_AlarmC := #AlarmC;
END_REGION

REGION Network 97: **** 9.1 - Alarm Output **** Alarm D
   // Alarm D
   #O_AlarmD := #AlarmD;
END_REGION

REGION Network 98: **** 9.2 - Alarm DWord**** Alarm To DWord
   // Alarm To Word
   IF "TRUE" THEN
       "LAlarmDword"(I_Alarm00 := #AA_MotorProtection,
                     I_Alarm01 := #AA_SafetySwitch,
                     I_Alarm02 := #AC_BodyNotInPos,
                     I_Alarm03 := #AB_TrfOutSetOverTime,
                     I_Alarm04 := #AB_TrfOutResOverTime,
                     I_Alarm05 := #AD_TrfInResInterlock,
                     I_Alarm06 := #AD_TrfOutSetInterlock,
                     I_Alarm07 := #AB_Alarm,
                     I_Alarm08 := #AD_Warning,
                     I_Alarm09 := #AD_TrfOutResInterlock,
                     I_Alarm10 := #AD_TrfInSetInterlock,
                     I_Alarm11 := #AB_BeltControlSetDet,
                     I_Alarm12 := #AB_BeltControlResDet,
                     I_Alarm13 := #AB_LSpeedDetMissing,
                     I_Alarm14 := #AC_TrfInStopped,
                     I_Alarm15 := #AC_StopDetSet,
                     I_Alarm16 := #AC_StopDetRes,
                     I_Alarm17 := #AC_LowSpdDetSet,
                     I_Alarm18 := #AC_LowSpdDetRes,
                     I_Alarm19 := #AA_NoBusControl,
                     I_Alarm20 := #AC_ConfigCalibrationAlm,
                     I_Alarm21 := #AD_CalibrationSetWarn,
                     I_Alarm22 := #AD_CalibrationResetWarn,
                     I_Alarm23 := #AB_STO,
                     I_Alarm24 := #AC_ConfigRampAlm,
                     I_Alarm25 := #AC_ConfigRampCalcAlm,
                     I_Alarm26 := #AD_MotionStop,
                     I_Alarm27 := "FALSE",
                     I_Alarm28 := "FALSE",
                     I_Alarm29 := "FALSE",
                     I_Alarm30 := "FALSE",
                     I_Alarm31 := "FALSE",
                     H_AlarmDWord => #H_AlarmDWord);
   END_IF;
END_REGION
END_FUNCTION_BLOCK
